KUKA KRL program: MyProgram_193().src

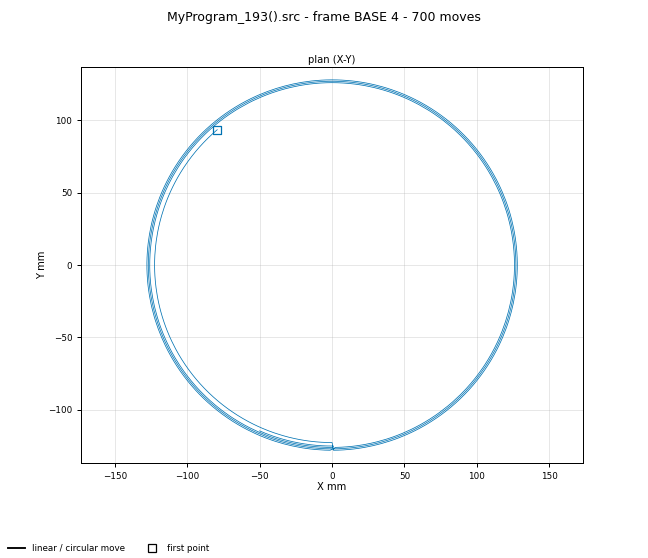
[picture p0: tool path of MyProgram_193().src in frame BASE 4, 700 of 700 moves have a stored position in this frame; points joined in program order, loops and branches not executed]
&ACCESS RVP
&REL 1
&PARAM TEMPLATE = C:\KRC\Roboter\Template\vorgabe
&PARAM EDITMASK = *
DEF MyProgram_193()
; ---- Setting reference (Base) ----
$BASE = BASE_DATA[4]

; --------------------------
; ---- Setting tool (TCP) ----
$TOOL = TOOL_DATA[3]
; --------------------------

$VEL.CP = VEL_APROX_PRINT
Startdeposition()
$VEL.CP = VEL_PRINT
LIN {X -79.3887,Y 93.5146,Z 139,A 127.081,B 23.6673,C -1.501,E1 23.6075,E2 679.4416} C_DIS
LIN {X -82.6375,Y 90.6569,Z 139,A 129.0803,B 23.6676,C -1.4955,E1 23.6034,E2 677.4477} C_DIS
LIN {X -85.6654,Y 87.8014,Z 139,A 131.1027,B 23.6676,C -1.4942,E1 23.5993,E2 675.4197} C_DIS
LIN {X -88.7871,Y 84.6429,Z 139,A 133.1305,B 23.6681,C -1.4871,E1 23.5954,E2 673.4002} C_DIS
LIN {X -91.627,Y 81.5608,Z 139,A 135.1651,B 23.6682,C -1.4854,E1 23.5916,E2 671.3603} C_DIS
LIN {X -94.341,Y 78.4052,Z 139,A 137.0999,B 23.6685,C -1.48,E1 23.5881,E2 669.4298} C_DIS
LIN {X -97.1692,Y 74.872,Z 139,A 139.2464,B 23.6688,C -1.4757,E1 23.5844,E2 667.2831} C_DIS
LIN {X -99.8211,Y 71.2973,Z 139,A 141.3446,B 23.6691,C -1.4708,E1 23.5809,E2 665.1863} C_DIS
LIN {X -102.4361,Y 67.4863,Z 139,A 143.4891,B 23.6694,C -1.4642,E1 23.5776,E2 663.047} C_DIS
LIN {X -104.8157,Y 63.7284,Z 139,A 145.6026,B 23.6697,C -1.4598,E1 23.5745,E2 660.9332} C_DIS
LIN {X -106.7407,Y 60.4493,Z 139,A 147.3793,B 23.67,C -1.4547,E1 23.572,E2 659.1594} C_DIS
LIN {X -108.6109,Y 57.0154,Z 139,A 149.1562,B 23.6704,C -1.4473,E1 23.5697,E2 657.391} C_DIS
LIN {X -110.2377,Y 53.8052,Z 139,A 150.913,B 23.6705,C -1.4454,E1 23.5675,E2 655.6289} C_DIS
LIN {X -111.8084,Y 50.4593,Z 139,A 152.53,B 23.6711,C -1.4356,E1 23.5657,E2 654.027} C_DIS
LIN {X -113.3266,Y 46.9501,Z 139,A 154.4547,B 23.6711,C -1.4359,E1 23.5636,E2 652.0901} C_DIS
LIN {X -114.6812,Y 43.5389,Z 139,A 156.1243,B 23.6715,C -1.4288,E1 23.5619,E2 650.4286} C_DIS
LIN {X -115.9983,Y 39.8949,Z 139,A 157.8402,B 23.672,C -1.4193,E1 23.5603,E2 648.7262} C_DIS
LIN {X -116.9413,Y 37.0399,Z 139,A 159.2538,B 23.6723,C -1.4152,E1 23.5591,E2 647.314} C_DIS
LIN {X -117.8141,Y 34.1624,Z 139,A 160.8056,B 23.6722,C -1.4169,E1 23.5578,E2 645.7485} C_DIS
LIN {X -118.9906,Y 29.8083,Z 139,A 162.938,B 23.6725,C -1.4113,E1 23.5563,E2 643.6172} C_DIS
LIN {X -119.8593,Y 26.095,Z 139,A 164.7128,B 23.6728,C -1.4053,E1 23.5553,E2 641.8462} C_DIS
LIN {X -120.5971,Y 22.4467,Z 139,A 166.3262,B 23.6734,C -1.3945,E1 23.5544,E2 640.2496} C_DIS
LIN {X -121.1103,Y 19.4926,Z 139,A 167.753,B 23.6736,C -1.3911,E1 23.5538,E2 638.8224} C_DIS
LIN {X -121.55,Y 16.5267,Z 139,A 169.2845,B 23.6736,C -1.392,E1 23.5532,E2 637.279} C_DIS
LIN {X -121.9936,Y 12.8387,Z 139,A 170.9072,B 23.6741,C -1.3817,E1 23.5527,E2 635.6716} C_DIS
LIN {X -122.2705,Y 9.8652,Z 139,A 172.3135,B 23.6743,C -1.3777,E1 23.5523,E2 634.2665} C_DIS
LIN {X -122.4784,Y 6.8343,Z 139,A 173.7573,B 23.6745,C -1.3741,E1 23.5521,E2 632.8224} C_DIS
LIN {X -122.6313,Y 2.9913,Z 139,A 175.5814,B 23.6748,C -1.3694,E1 23.5519,E2 630.9984} C_DIS
LIN {X -122.6672,Y -0.3879,Z 139,A 177.2488,B 23.6748,C -1.368,E1 23.5519,E2 629.324} C_DIS
LIN {X -122.5842,Y -4.5164,Z 139,A 179.0836,B 23.6754,C -1.3579,E1 23.552,E2 627.5027} C_DIS
LIN {X -122.44,Y -7.4601,Z 139,A -179.4399,B 23.6754,C -1.3576,E1 23.5523,E2 626.0175} C_DIS
LIN {X -122.1123,Y -11.6529,Z 139,A -177.4861,B 23.6758,C -1.3509,E1 23.5527,E2 624.0681} C_DIS
LIN {X -121.6563,Y -15.7152,Z 139,A -175.6057,B 23.6762,C -1.3436,E1 23.5534,E2 622.1941} C_DIS
LIN {X -121.2209,Y -18.7791,Z 139,A -174.1758,B 23.6765,C -1.3383,E1 23.5539,E2 620.7682} C_DIS
LIN {X -120.73,Y -21.7125,Z 139,A -172.7657,B 23.6767,C -1.3348,E1 23.5546,E2 619.358} C_DIS
LIN {X -120.0095,Y -25.3991,Z 139,A -170.9856,B 23.6769,C -1.3304,E1 23.5556,E2 617.5779} C_DIS
LIN {X -119.1851,Y -29.0196,Z 139,A -169.2623,B 23.6772,C -1.3246,E1 23.5567,E2 615.8584} C_DIS
LIN {X -118.4092,Y -32.0405,Z 139,A -167.6338,B 23.6771,C -1.3272,E1 23.5579,E2 614.2133} C_DIS
LIN {X -117.3595,Y -35.6921,Z 139,A -166.0055,B 23.6777,C -1.3157,E1 23.5592,E2 612.6037} C_DIS
LIN {X -116.2196,Y -39.248,Z 139,A -164.0849,B 23.6776,C -1.3178,E1 23.5608,E2 610.6662} C_DIS
LIN {X -114.9815,Y -42.7371,Z 139,A -162.5098,B 23.6782,C -1.3062,E1 23.5623,E2 609.1106} C_DIS
LIN {X -113.8941,Y -45.556,Z 139,A -160.9775,B 23.6782,C -1.3072,E1 23.5639,E2 607.567} C_DIS
LIN {X -112.4784,Y -48.9468,Z 139,A -159.3454,B 23.6786,C -1.2987,E1 23.5657,E2 605.9466} C_DIS
LIN {X -110.9144,Y -52.3963,Z 139,A -157.5959,B 23.6789,C -1.2928,E1 23.5677,E2 604.2016} C_DIS
LIN {X -109.5682,Y -55.1562,Z 139,A -156.145,B 23.679,C -1.2895,E1 23.5695,E2 602.7507} C_DIS
LIN {X -108.185,Y -57.824,Z 139,A -154.585,B 23.6789,C -1.2921,E1 23.5716,E2 601.1753} C_DIS
LIN {X -105.9858,Y -61.7632,Z 139,A -152.4677,B 23.6792,C -1.2868,E1 23.5745,E2 599.0594} C_DIS
LIN {X -104.0005,Y -65.0502,Z 139,A -150.6485,B 23.6793,C -1.2832,E1 23.5772,E2 597.2395} C_DIS
LIN {X -101.5455,Y -68.819,Z 139,A -148.5147,B 23.6796,C -1.2792,E1 23.5805,E2 595.1044} C_DIS
LIN {X -98.9417,Y -72.5127,Z 139,A -146.4248,B 23.6799,C -1.273,E1 23.5839,E2 593.0191} C_DIS
LIN {X -96.2459,Y -76.0552,Z 139,A -144.3049,B 23.68,C -1.2697,E1 23.5875,E2 590.8969} C_DIS
LIN {X -93.644,Y -79.2365,Z 139,A -142.5065,B 23.6805,C -1.26,E1 23.5907,E2 589.1139} C_DIS
LIN {X -91.1571,Y -82.0855,Z 139,A -140.6177,B 23.6805,C -1.2612,E1 23.5942,E2 587.2131} C_DIS
LIN {X -88.24,Y -85.2131,Z 139,A -138.6381,B 23.6807,C -1.256,E1 23.598,E2 585.2373} C_DIS
LIN {X -85.1287,Y -88.3217,Z 139,A -136.6069,B 23.681,C -1.2507,E1 23.6021,E2 583.2104} C_DIS
LIN {X -82.1159,Y -91.1299,Z 139,A -134.5975,B 23.681,C -1.2504,E1 23.6062,E2 581.193} C_DIS
LIN {X -78.7723,Y -94.0344,Z 139,A -132.6267,B 23.6814,C -1.2422,E1 23.6104,E2 579.2346} C_DIS
LIN {X -75.7059,Y -96.5203,Z 139,A -130.7809,B 23.6816,C -1.2389,E1 23.6144,E2 577.3898} C_DIS
LIN {X -72.5193,Y -98.9369,Z 139,A -128.955,B 23.6818,C -1.2338,E1 23.6185,E2 575.5698} C_DIS
LIN {X -69.4074,Y -101.1442,Z 139,A -127.0058,B 23.6816,C -1.238,E1 23.623,E2 573.6029} C_DIS
LIN {X -65.6311,Y -103.6346,Z 139,A -124.9026,B 23.6818,C -1.2343,E1 23.6279,E2 571.5018} C_DIS
LIN {X -61.7652,Y -105.9846,Z 139,A -122.7608,B 23.6818,C -1.2324,E1 23.6331,E2 569.3578} C_DIS
LIN {X -57.8305,Y -108.1816,Z 139,A -120.6273,B 23.682,C -1.2308,E1 23.6383,E2 567.2219} C_DIS
LIN {X -54.5438,Y -109.8734,Z 139,A -119.0576,B 23.6824,C -1.2218,E1 23.6422,E2 565.6702} C_DIS
LIN {X -51.5071,Y -111.3288,Z 139,A -117.4725,B 23.6824,C -1.2205,E1 23.6462,E2 564.0843} C_DIS
LIN {X -48.3233,Y -112.748,Z 139,A -115.7041,B 23.6823,C -1.2249,E1 23.6507,E2 562.3005} C_DIS
LIN {X -44.1464,Y -114.4478,Z 139,A -113.6361,B 23.6824,C -1.2211,E1 23.6561,E2 560.237} C_DIS
LIN {X -39.9096,Y -115.9932,Z 139,A -111.6551,B 23.6828,C -1.2137,E1 23.6613,E2 558.2704} C_DIS
LIN {X -37.055,Y -116.9364,Z 139,A -110.2492,B 23.6828,C -1.2126,E1 23.665,E2 556.8643} C_DIS
LIN {X -34.1778,Y -117.8096,Z 139,A -108.7044,B 23.6826,C -1.2179,E1 23.6692,E2 555.3038} C_DIS
LIN {X -29.8197,Y -118.9876,Z 139,A -106.5916,B 23.6826,C -1.2168,E1 23.6749,E2 553.1904} C_DIS
LIN {X -25.9912,Y -119.8817,Z 139,A -104.7935,B 23.6828,C -1.2142,E1 23.6798,E2 551.3964} C_DIS
LIN {X -22.4579,Y -120.595,Z 139,A -103.0548,B 23.6827,C -1.216,E1 23.6846,E2 549.6512} C_DIS
LIN {X -18.7973,Y -121.2181,Z 139,A -101.4495,B 23.683,C -1.2097,E1 23.6889,E2 548.0601} C_DIS
LIN {X -15.7039,Y -121.6578,Z 139,A -99.8752,B 23.6828,C -1.2145,E1 23.6933,E2 546.4724} C_DIS
LIN {X -11.2234,Y -122.1535,Z 139,A -97.7609,B 23.6828,C -1.2147,E1 23.6992,E2 544.3564} C_DIS
LIN {X -7.5226,Y -122.4362,Z 139,A -96.1117,B 23.6829,C -1.2109,E1 23.7038,E2 542.7161} C_DIS
LIN {X -3.7044,Y -122.6115,Z 139,A -94.259,B 23.6828,C -1.2141,E1 23.709,E2 540.855} C_DIS
LIN {X -0.005,Y -122.669,Z 139,A -92.6349,B 23.683,C -1.2097,E1 23.7135,E2 539.2418} C_DIS
LIN {X -0.005,Y -122.669,Z 139,A -92.6349,B 23.683,C -1.2097,E1 23.7135,E2 539.2418} C_DIS
Enddeposition()
LIN {X 0.9076,Y -127.9731,Z 140,A -92.6066,B 24.9649,C -1.3697,E1 25.0021,E2 539.0016} C_DIS
Startdeposition()
$VEL.CP = VEL_PRINT
LIN {X 4.2701,Y -127.9089,Z 140,A -90.8609,B 24.9642,C -1.3823,E1 25.0071,E2 537.2265} C_DIS
LIN {X 8.0025,Y -127.7277,Z 140,A -89.2685,B 24.9644,C -1.3789,E1 25.0115,E2 535.6426} C_DIS
LIN {X 12.0529,Y -127.4094,Z 140,A -87.5467,B 24.9646,C -1.3749,E1 25.0162,E2 533.9312} C_DIS
LIN {X 14.9814,Y -127.0982,Z 140,A -86.1517,B 24.9643,C -1.3796,E1 25.0201,E2 532.5262} C_DIS
LIN {X 18.2831,Y -126.6654,Z 140,A -84.6512,B 24.9643,C -1.3811,E1 25.0243,E2 531.0233} C_DIS
LIN {X 22.3408,Y -126.013,Z 140,A -82.8669,B 24.9643,C -1.3797,E1 25.0292,E2 529.2443} C_DIS
LIN {X 25.4642,Y -125.419,Z 140,A -81.4803,B 24.9643,C -1.379,E1 25.033,E2 527.8608} C_DIS
LIN {X 28.3673,Y -124.7944,Z 140,A -80.2161,B 24.9645,C -1.3769,E1 25.0364,E2 526.6033} C_DIS
LIN {X 31.3018,Y -124.0909,Z 140,A -78.771,B 24.9642,C -1.3831,E1 25.0404,E2 525.1456} C_DIS
LIN {X 34.2875,Y -123.2993,Z 140,A -77.4974,B 24.9644,C -1.379,E1 25.0438,E2 523.8838} C_DIS
LIN {X 37.2721,Y -122.4301,Z 140,A -76.2359,B 24.9646,C -1.3739,E1 25.0471,E2 522.6365} C_DIS
LIN {X 40.0928,Y -121.536,Z 140,A -74.6318,B 24.9638,C -1.3899,E1 25.0515,E2 520.9976} C_DIS
LIN {X 43.2265,Y -120.4567,Z 140,A -73.2401,B 24.964,C -1.3871,E1 25.0551,E2 519.6153} C_DIS
LIN {X 46.1903,Y -119.3515,Z 140,A -71.7808,B 24.9637,C -1.3913,E1 25.0589,E2 518.1492} C_DIS
LIN {X 49.1413,Y -118.1671,Z 140,A -70.3614,B 24.9637,C -1.3932,E1 25.0626,E2 516.7287} C_DIS
LIN {X 51.9549,Y -116.9576,Z 140,A -69.1813,B 24.964,C -1.3854,E1 25.0656,E2 515.5699} C_DIS
LIN {X 54.9013,Y -115.6037,Z 140,A -67.5632,B 24.9635,C -1.3963,E1 25.0697,E2 513.9301} C_DIS
LIN {X 57.8129,Y -114.1754,Z 140,A -66.0746,B 24.9633,C -1.4007,E1 25.0735,E2 512.4352} C_DIS
LIN {X 60.9283,Y -112.5463,Z 140,A -64.3996,B 24.9628,C -1.4087,E1 25.0776,E2 510.746} C_DIS
LIN {X 64.6643,Y -110.4415,Z 140,A -62.4971,B 24.9627,C -1.4113,E1 25.0822,E2 508.843} C_DIS
LIN {X 68.3933,Y -108.1717,Z 140,A -60.6188,B 24.9627,C -1.4111,E1 25.0867,E2 506.9712} C_DIS
LIN {X 71.8212,Y -105.9268,Z 140,A -58.7909,B 24.9625,C -1.4145,E1 25.0909,E2 505.1415} C_DIS
LIN {X 75.297,Y -103.4851,Z 140,A -56.8856,B 24.9623,C -1.4186,E1 25.0953,E2 503.233} C_DIS
LIN {X 78.6223,Y -100.982,Z 140,A -54.9796,B 24.962,C -1.425,E1 25.0995,E2 501.3189} C_DIS
LIN {X 81.9467,Y -98.3039,Z 140,A -53.0464,B 24.9617,C -1.4304,E1 25.1037,E2 499.3801} C_DIS
LIN {X 85.2482,Y -95.4543,Z 140,A -51.1346,B 24.9615,C -1.4329,E1 25.1077,E2 497.4702} C_DIS
LIN {X 88.4654,Y -92.4804,Z 140,A -49.1994,B 24.9614,C -1.4363,E1 25.1116,E2 495.535} C_DIS
LIN {X 91.6345,Y -89.3421,Z 140,A -47.1815,B 24.961,C -1.4424,E1 25.1156,E2 493.5112} C_DIS
LIN {X 94.5006,Y -86.305,Z 140,A -45.3542,B 24.9609,C -1.4449,E1 25.1191,E2 491.686} C_DIS
LIN {X 97.2409,Y -83.2054,Z 140,A -43.4679,B 24.9605,C -1.4516,E1 25.1225,E2 489.7924} C_DIS
LIN {X 100.0412,Y -79.8156,Z 140,A -41.547,B 24.9604,C -1.4544,E1 25.1259,E2 487.8738} C_DIS
LIN {X 102.646,Y -76.4365,Z 140,A -39.6801,B 24.9602,C -1.4574,E1 25.129,E2 486.0088} C_DIS
LIN {X 105.1099,Y -73.0114,Z 140,A -37.8242,B 24.96,C -1.461,E1 25.132,E2 484.1535} C_DIS
LIN {X 107.2878,Y -69.7717,Z 140,A -36.0336,B 24.9596,C -1.4683,E1 25.1348,E2 482.3546} C_DIS
LIN {X 109.6772,Y -65.9528,Z 140,A -34.1134,B 24.9596,C -1.469,E1 25.1376,E2 480.4424} C_DIS
LIN {X 111.6754,Y -62.5093,Z 140,A -32.2598,B 24.9591,C -1.4781,E1 25.1402,E2 478.5769} C_DIS
LIN {X 113.7807,Y -58.5882,Z 140,A -30.3362,B 24.9589,C -1.4805,E1 25.1427,E2 476.658} C_DIS
LIN {X 115.1293,Y -55.8943,Z 140,A -29.0433,B 24.9589,C -1.4816,E1 25.1443,E2 475.3694} C_DIS
LIN {X 116.4969,Y -52.9848,Z 140,A -27.6149,B 24.9587,C -1.4854,E1 25.1459,E2 473.9396} C_DIS
LIN {X 117.9777,Y -49.5948,Z 140,A -25.9435,B 24.9583,C -1.4914,E1 25.1478,E2 472.2632} C_DIS
LIN {X 119.233,Y -46.4952,Z 140,A -24.5,B 24.9583,C -1.4933,E1 25.1493,E2 470.8233} C_DIS
LIN {X 120.2222,Y -43.8768,Z 140,A -23.1739,B 24.9578,C -1.5011,E1 25.1506,E2 469.4861} C_DIS
LIN {X 121.1957,Y -41.1148,Z 140,A -21.8125,B 24.9574,C -1.508,E1 25.1518,E2 468.1162} C_DIS
LIN {X 122.3197,Y -37.6329,Z 140,A -20.3174,B 24.9575,C -1.5056,E1 25.1531,E2 466.6353} C_DIS
LIN {X 123.2027,Y -34.6331,Z 140,A -19.0434,B 24.9577,C -1.5034,E1 25.154,E2 465.3737} C_DIS
LIN {X 123.8556,Y -32.229,Z 140,A -17.7303,B 24.9569,C -1.5176,E1 25.155,E2 464.0348} C_DIS
LIN {X 124.5942,Y -29.2441,Z 140,A -16.3459,B 24.9566,C -1.5225,E1 25.1559,E2 462.6469} C_DIS
LIN {X 125.2565,Y -26.2628,Z 140,A -14.9625,B 24.9563,C -1.5278,E1 25.1567,E2 461.259} C_DIS
LIN {X 125.9442,Y -22.7253,Z 140,A -13.4705,B 24.9563,C -1.5266,E1 25.1574,E2 459.7785} C_DIS
LIN {X 126.4433,Y -19.761,Z 140,A -12.168,B 24.9563,C -1.5287,E1 25.158,E2 458.4787} C_DIS
LIN {X 126.8932,Y -16.6281,Z 140,A -10.7317,B 24.9559,C -1.5344,E1 25.1586,E2 457.0375} C_DIS
LIN {X 127.3223,Y -12.9601,Z 140,A -8.9614,B 24.9552,C -1.5461,E1 25.1591,E2 455.2501} C_DIS
LIN {X 127.6326,Y -9.3972,Z 140,A -7.5269,B 24.9554,C -1.5425,E1 25.1594,E2 453.8326} C_DIS
LIN {X 127.8325,Y -6.1114,Z 140,A -5.9091,B 24.9547,C -1.5551,E1 25.1597,E2 452.1947} C_DIS
LIN {X 127.9576,Y -2.3014,Z 140,A -4.346,B 24.9548,C -1.553,E1 25.1597,E2 450.6458} C_DIS
LIN {X 127.9704,Y 1.5309,Z 140,A -2.5591,B 24.9543,C -1.5624,E1 25.1597,E2 448.8473} C_DIS
LIN {X 127.8741,Y 5.1617,Z 140,A -1.0017,B 24.9542,C -1.5641,E1 25.1597,E2 447.2952} C_DIS
LIN {X 127.6513,Y 9.1421,Z 140,A 0.7262,B 24.954,C -1.5669,E1 25.1593,E2 445.5709} C_DIS
LIN {X 127.4094,Y 12.0529,Z 140,A 2.0613,B 24.9537,C -1.5727,E1 25.159,E2 444.2302} C_DIS
LIN {X 127.0363,Y 15.5009,Z 140,A 3.7184,B 24.953,C -1.5833,E1 25.1584,E2 442.5579} C_DIS
LIN {X 126.5623,Y 18.9921,Z 140,A 5.2467,B 24.9529,C -1.5857,E1 25.1578,E2 441.0329} C_DIS
LIN {X 126.0297,Y 22.2478,Z 140,A 6.6306,B 24.9529,C -1.5855,E1 25.1572,E2 439.6575} C_DIS
LIN {X 125.4446,Y 25.3382,Z 140,A 8.0006,B 24.9528,C -1.588,E1 25.1564,E2 438.2898} C_DIS
LIN {X 124.7727,Y 28.4626,Z 140,A 9.3377,B 24.9528,C -1.5875,E1 25.1556,E2 436.9615} C_DIS
LIN {X 124.0864,Y 31.3198,Z 140,A 10.7285,B 24.9523,C -1.5957,E1 25.1547,E2 435.5595} C_DIS
LIN {X 123.04,Y 35.2148,Z 140,A 12.5291,B 24.952,C -1.601,E1 25.1534,E2 433.7568} C_DIS
LIN {X 122.1223,Y 38.2746,Z 140,A 14.0391,B 24.9515,C -1.6097,E1 25.1521,E2 432.2349} C_DIS
LIN {X 120.9796,Y 41.7406,Z 140,A 15.5777,B 24.9515,C -1.6097,E1 25.1507,E2 430.705} C_DIS
LIN {X 119.9332,Y 44.6586,Z 140,A 16.9722,B 24.9512,C -1.6142,E1 25.1494,E2 429.3076} C_DIS
LIN {X 118.7692,Y 47.6676,Z 140,A 18.3953,B 24.951,C -1.6173,E1 25.1479,E2 427.885} C_DIS
LIN {X 117.5887,Y 50.5101,Z 140,A 19.5686,B 24.9514,C -1.6106,E1 25.1467,E2 426.7341} C_DIS
LIN {X 116.282,Y 53.4496,Z 140,A 21.2237,B 24.9505,C -1.6261,E1 25.1448,E2 425.0513} C_DIS
LIN {X 114.8656,Y 56.4288,Z 140,A 22.6722,B 24.9503,C -1.6289,E1 25.143,E2 423.604} C_DIS
LIN {X 113.3976,Y 59.3236,Z 140,A 24.1224,B 24.95,C -1.6328,E1 25.1412,E2 422.1522} C_DIS
LIN {X 111.366,Y 63.0599,Z 140,A 26.1237,B 24.9494,C -1.6432,E1 25.1384,E2 420.1368} C_DIS
LIN {X 109.3021,Y 66.5731,Z 140,A 27.9392,B 24.9491,C -1.6477,E1 25.1358,E2 418.32} C_DIS
LIN {X 107.0663,Y 70.1118,Z 140,A 29.8057,B 24.9488,C -1.6523,E1 25.133,E2 416.4521} C_DIS
LIN {X 104.6388,Y 73.685,Z 140,A 31.7003,B 24.9487,C -1.6552,E1 25.13,E2 414.5599} C_DIS
LIN {X 102.0732,Y 77.2,Z 140,A 33.6298,B 24.9484,C -1.6592,E1 25.1268,E2 412.6303} C_DIS
LIN {X 99.4073,Y 80.6043,Z 140,A 35.5612,B 24.9481,C -1.6637,E1 25.1234,E2 410.6974} C_DIS
LIN {X 96.7011,Y 83.8321,Z 140,A 37.495,B 24.9477,C -1.6706,E1 25.1199,E2 408.7559} C_DIS
LIN {X 93.9403,Y 86.9146,Z 140,A 39.2777,B 24.9477,C -1.6712,E1 25.1165,E2 406.9797} C_DIS
LIN {X 91.0503,Y 89.9374,Z 140,A 41.1467,B 24.9474,C -1.6752,E1 25.1129,E2 405.1093} C_DIS
LIN {X 88.1229,Y 92.8077,Z 140,A 43.0115,B 24.9471,C -1.6807,E1 25.1091,E2 403.2393} C_DIS
LIN {X 85.0157,Y 95.6619,Z 140,A 44.9026,B 24.9468,C -1.6847,E1 25.1052,E2 401.3464} C_DIS
LIN {X 81.942,Y 98.3079,Z 140,A 46.6565,B 24.9468,C -1.685,E1 25.1015,E2 399.5985} C_DIS
LIN {X 78.7277,Y 100.9003,Z 140,A 48.5386,B 24.9465,C -1.6902,E1 25.0974,E2 397.711} C_DIS
LIN {X 75.345,Y 103.4503,Z 140,A 50.4087,B 24.9463,C -1.6923,E1 25.0932,E2 395.8428} C_DIS
LIN {X 71.9763,Y 105.8218,Z 140,A 52.2755,B 24.9461,C -1.6966,E1 25.0889,E2 393.9722} C_DIS
LIN {X 68.0587,Y 108.3829,Z 140,A 54.3229,B 24.9461,C -1.6975,E1 25.0841,E2 391.9294} C_DIS
LIN {X 64.4713,Y 110.5548,Z 140,A 56.2279,B 24.9457,C -1.7017,E1 25.0795,E2 390.0203} C_DIS
LIN {X 60.7747,Y 112.6288,Z 140,A 58.1089,B 24.9457,C -1.7035,E1 25.0749,E2 388.1404} C_DIS
LIN {X 57.1568,Y 114.5065,Z 140,A 59.901,B 24.9456,C -1.7043,E1 25.0704,E2 386.3514} C_DIS
LIN {X 53.8901,Y 116.0783,Z 140,A 61.4268,B 24.9458,C -1.7013,E1 25.0666,E2 384.8365} C_DIS
LIN {X 50.0553,Y 117.7854,Z 140,A 63.433,B 24.9452,C -1.7099,E1 25.0614,E2 382.815} C_DIS
LIN {X 46.6151,Y 119.1864,Z 140,A 64.9753,B 24.9455,C -1.7055,E1 25.0575,E2 381.2865} C_DIS
LIN {X 43.5103,Y 120.3543,Z 140,A 66.2806,B 24.946,C -1.6978,E1 25.0541,E2 380.0021} C_DIS
LIN {X 41.1775,Y 121.1748,Z 140,A 67.6036,B 24.9452,C -1.7097,E1 25.0505,E2 378.6537} C_DIS
LIN {X 37.8444,Y 122.255,Z 140,A 69.164,B 24.9452,C -1.7105,E1 25.0464,E2 377.0941} C_DIS
LIN {X 34.5678,Y 123.2209,Z 140,A 70.6014,B 24.9454,C -1.707,E1 25.0425,E2 375.6674} C_DIS
LIN {X 30.3415,Y 124.3296,Z 140,A 72.4573,B 24.9456,C -1.7032,E1 25.0376,E2 373.8234} C_DIS
LIN {X 27.2217,Y 125.0495,Z 140,A 74.0505,B 24.9451,C -1.712,E1 25.0332,E2 372.2116} C_DIS
LIN {X 24.0369,Y 125.7003,Z 140,A 75.4916,B 24.9451,C -1.712,E1 25.0292,E2 370.7724} C_DIS
LIN {X 20.7847,Y 126.2792,Z 140,A 77.0061,B 24.9449,C -1.7142,E1 25.025,E2 369.254} C_DIS
LIN {X 16.8085,Y 126.8695,Z 140,A 78.7456,B 24.9451,C -1.7117,E1 25.0203,E2 367.522} C_DIS
LIN {X 13.7363,Y 127.2387,Z 140,A 80.1561,B 24.945,C -1.7132,E1 25.0163,E2 366.109} C_DIS
LIN {X 10.0436,Y 127.5855,Z 140,A 81.9323,B 24.9446,C -1.719,E1 25.0114,E2 364.3199} C_DIS
LIN {X 6.6351,Y 127.8062,Z 140,A 83.3074,B 24.9451,C -1.7114,E1 25.0076,E2 362.9633} C_DIS
LIN {X 3.3822,Y 127.9336,Z 140,A 84.8526,B 24.9448,C -1.7156,E1 25.0032,E2 361.4085} C_DIS
LIN {X -0.5369,Y 127.9772,Z 140,A 86.5777,B 24.945,C -1.7139,E1 24.9984,E2 359.6877} C_DIS
LIN {X -4.2701,Y 127.9089,Z 140,A 88.3434,B 24.9447,C -1.718,E1 24.9935,E2 357.9121} C_DIS
LIN {X -7.3727,Y 127.7665,Z 140,A 89.6721,B 24.9449,C -1.7144,E1 24.9898,E2 356.5914} C_DIS
LIN {X -10.6356,Y 127.5354,Z 140,A 91.1001,B 24.9451,C -1.712,E1 24.9858,E2 355.1686} C_DIS
LIN {X -14.425,Y 127.1646,Z 140,A 92.7573,B 24.9453,C -1.7087,E1 24.9813,E2 353.5182} C_DIS
LIN {X -17.9065,Y 126.7192,Z 140,A 94.2585,B 24.9456,C -1.7044,E1 24.9771,E2 352.0262} C_DIS
LIN {X -20.8827,Y 126.2628,Z 140,A 95.6821,B 24.9454,C -1.7071,E1 24.9732,E2 350.5949} C_DIS
LIN {X -23.8508,Y 125.7359,Z 140,A 97.0402,B 24.9454,C -1.7064,E1 24.9694,E2 349.2369} C_DIS
LIN {X -26.8272,Y 125.1346,Z 140,A 98.4043,B 24.9454,C -1.7055,E1 24.9657,E2 347.8734} C_DIS
LIN {X -29.8344,Y 124.4519,Z 140,A 99.7833,B 24.9456,C -1.7041,E1 24.962,E2 346.4958} C_DIS
LIN {X -32.7946,Y 123.7048,Z 140,A 101.1615,B 24.9456,C -1.7033,E1 24.9582,E2 345.1175} C_DIS
LIN {X -35.8577,Y 122.8518,Z 140,A 102.5709,B 24.9458,C -1.7011,E1 24.9545,E2 343.7112} C_DIS
LIN {X -38.6322,Y 122.0081,Z 140,A 103.9297,B 24.9457,C -1.7025,E1 24.9508,E2 342.3467} C_DIS
LIN {X -41.7684,Y 120.97,Z 140,A 105.389,B 24.9459,C -1.6997,E1 24.947,E2 340.8912} C_DIS
LIN {X -44.5407,Y 119.9773,Z 140,A 106.7502,B 24.9459,C -1.7,E1 24.9434,E2 339.5266} C_DIS
LIN {X -47.7395,Y 118.7402,Z 140,A 108.225,B 24.9462,C -1.695,E1 24.9396,E2 338.0604} C_DIS
LIN {X -50.3417,Y 117.6615,Z 140,A 109.554,B 24.9461,C -1.6964,E1 24.9362,E2 336.7251} C_DIS
LIN {X -53.2438,Y 116.3772,Z 140,A 110.8221,B 24.9467,C -1.6869,E1 24.933,E2 335.4765} C_DIS
LIN {X -56.2714,Y 114.9433,Z 140,A 112.4688,B 24.9464,C -1.6915,E1 24.9288,E2 333.8146} C_DIS
LIN {X -59.3236,Y 113.3976,Z 140,A 113.9543,B 24.9467,C -1.6867,E1 24.9251,E2 332.3363} C_DIS
LIN {X -62.81,Y 111.5064,Z 140,A 115.8077,B 24.9467,C -1.6873,E1 24.9206,E2 330.4764} C_DIS
LIN {X -66.4172,Y 109.3963,Z 140,A 117.7249,B 24.9467,C -1.686,E1 24.916,E2 328.5563} C_DIS
LIN {X -70.0382,Y 107.1147,Z 140,A 119.7053,B 24.9467,C -1.6853,E1 24.9113,E2 326.5711} C_DIS
LIN {X -73.5809,Y 104.7122,Z 140,A 121.6148,B 24.947,C -1.6811,E1 24.9069,E2 324.6652} C_DIS
LIN {X -77.1713,Y 102.0948,Z 140,A 123.5505,B 24.9475,C -1.6744,E1 24.9026,E2 322.7387} C_DIS
LIN {X -80.4221,Y 99.5542,Z 140,A 125.3987,B 24.9477,C -1.6704,E1 24.8986,E2 320.8931} C_DIS
LIN {X -83.5947,Y 96.9056,Z 140,A 127.2585,B 24.9479,C -1.6666,E1 24.8946,E2 319.035} C_DIS
LIN {X -86.6873,Y 94.1492,Z 140,A 129.122,B 24.9482,C -1.6627,E1 24.8908,E2 317.1735} C_DIS
LIN {X -89.684,Y 91.2991,Z 140,A 130.9841,B 24.9484,C -1.6587,E1 24.887,E2 315.3131} C_DIS
LIN {X -92.5909,Y 88.3497,Z 140,A 132.8534,B 24.9487,C -1.6548,E1 24.8834,E2 313.4451} C_DIS
LIN {X -95.4919,Y 85.2062,Z 140,A 134.8134,B 24.9489,C -1.652,E1 24.8797,E2 311.4831} C_DIS
LIN {X -98.3241,Y 81.9224,Z 140,A 136.7747,B 24.9491,C -1.6478,E1 24.8762,E2 309.5228} C_DIS
LIN {X -100.9003,Y 78.7277,Z 140,A 138.6622,B 24.9493,C -1.6451,E1 24.8729,E2 307.6326} C_DIS
LIN {X -103.4625,Y 75.3282,Z 140,A 140.5726,B 24.9496,C -1.6401,E1 24.8697,E2 305.7251} C_DIS
LIN {X -106.0437,Y 71.6484,Z 140,A 142.5286,B 24.9501,C -1.6318,E1 24.8666,E2 303.7792} C_DIS
LIN {X -108.3591,Y 68.0965,Z 140,A 144.4735,B 24.9503,C -1.6285,E1 24.8637,E2 301.8322} C_DIS
LIN {X -110.5548,Y 64.4713,Z 140,A 146.3991,B 24.9506,C -1.6243,E1 24.861,E2 299.9069} C_DIS
LIN {X -112.5462,Y 60.9283,Z 140,A 148.2396,B 24.9508,C -1.6198,E1 24.8585,E2 298.0672} C_DIS
LIN {X -114.4159,Y 57.3405,Z 140,A 149.9697,B 24.9514,C -1.6106,E1 24.8563,E2 296.3499} C_DIS
LIN {X -116.0186,Y 54.0192,Z 140,A 151.6307,B 24.9517,C -1.606,E1 24.8543,E2 294.6907} C_DIS
LIN {X -117.7854,Y 50.0553,Z 140,A 153.653,B 24.9518,C -1.6037,E1 24.8521,E2 292.6629} C_DIS
LIN {X -119.1516,Y 46.7046,Z 140,A 155.2204,B 24.9523,C -1.5962,E1 24.8505,E2 291.1045} C_DIS
LIN {X -120.3018,Y 43.6561,Z 140,A 156.5299,B 24.9529,C -1.5847,E1 24.8492,E2 289.815} C_DIS
LIN {X -121.2998,Y 40.8021,Z 140,A 158.0572,B 24.9527,C -1.5884,E1 24.8478,E2 288.2701} C_DIS
LIN {X -122.1466,Y 38.1986,Z 140,A 159.237,B 24.9531,C -1.5824,E1 24.8468,E2 287.0981} C_DIS
LIN {X -123.1836,Y 34.7013,Z 140,A 160.9106,B 24.9533,C -1.579,E1 24.8455,E2 285.4227} C_DIS
LIN {X -124.3118,Y 30.4156,Z 140,A 162.933,B 24.9536,C -1.5744,E1 24.8441,E2 283.3996} C_DIS
LIN {X -125.0286,Y 27.3181,Z 140,A 164.1866,B 24.9543,C -1.5619,E1 24.8434,E2 282.1684} C_DIS
LIN {X -125.6619,Y 24.2378,Z 140,A 165.7268,B 24.9543,C -1.5634,E1 24.8425,E2 280.6155} C_DIS
LIN {X -126.2167,Y 21.1594,Z 140,A 167.1076,B 24.9545,C -1.5579,E1 24.8418,E2 279.2396} C_DIS
LIN {X -126.6966,Y 18.0649,Z 140,A 168.4879,B 24.9549,C -1.5523,E1 24.8413,E2 277.8644} C_DIS
LIN {X -127.0621,Y 15.2845,Z 140,A 169.7862,B 24.9549,C -1.5502,E1 24.8408,E2 276.5635} C_DIS
LIN {X -127.3821,Y 12.3363,Z 140,A 171.1888,B 24.955,C -1.5493,E1 24.8404,E2 275.1546} C_DIS
LIN {X -127.6914,Y 8.5924,Z 140,A 172.888,B 24.9553,C -1.5445,E1 24.8401,E2 273.4565} C_DIS
LIN {X -127.8741,Y 5.1617,Z 140,A 174.4403,B 24.9556,C -1.5401,E1 24.8399,E2 271.9053} C_DIS
LIN {X -127.9723,Y 1.4172,Z 140,A 176.0883,B 24.956,C -1.5332,E1 24.8398,E2 270.2638} C_DIS
LIN {X -127.9536,Y -2.5439,Z 140,A 177.9563,B 24.956,C -1.5318,E1 24.8398,E2 268.3879} C_DIS
LIN {X -127.8255,Y -6.2512,Z 140,A 179.581,B 24.9564,C -1.5247,E1 24.84,E2 266.7703} C_DIS
LIN {X -127.5834,Y -10.0675,Z 140,A -178.5933,B 24.9564,C -1.5244,E1 24.8404,E2 264.9345} C_DIS
LIN {X -127.2627,Y -13.5137,Z 140,A -177.1468,B 24.957,C -1.5146,E1 24.8408,E2 263.5027} C_DIS
LIN {X -126.8695,Y -16.8085,Z 140,A -175.6162,B 24.9572,C -1.5119,E1 24.8413,E2 261.9694} C_DIS
LIN {X -126.2628,Y -20.8827,Z 140,A -173.8309,B 24.9577,C -1.5032,E1 24.8421,E2 260.1941} C_DIS
LIN {X -125.7359,Y -23.8508,Z 140,A -172.4692,B 24.9579,C -1.4995,E1 24.8428,E2 258.8333} C_DIS
LIN {X -125.1345,Y -26.8277,Z 140,A -171.0613,B 24.9579,C -1.4974,E1 24.8436,E2 257.422} C_DIS
LIN {X -124.4947,Y -29.6568,Z 140,A -169.7473,B 24.9582,C -1.494,E1 24.8444,E2 256.1083} C_DIS
LIN {X -123.6844,Y -32.8711,Z 140,A -168.3119,B 24.9586,C -1.4871,E1 24.8454,E2 254.681} C_DIS
LIN {X -122.8897,Y -35.7281,Z 140,A -166.9404,B 24.9586,C -1.485,E1 24.8465,E2 253.3066} C_DIS
LIN {X -122.113,Y -38.3039,Z 140,A -165.7853,B 24.959,C -1.479,E1 24.8474,E2 252.1591} C_DIS
LIN {X -121.0229,Y -41.6156,Z 140,A -164.1324,B 24.959,C -1.4786,E1 24.8489,E2 250.4979} C_DIS
LIN {X -120.1242,Y -44.1485,Z 140,A -162.83,B 24.959,C -1.4795,E1 24.8502,E2 249.1858} C_DIS
LIN {X -118.7692,Y -47.6676,Z 140,A -161.2539,B 24.9596,C -1.4693,E1 24.8518,E2 247.6252} C_DIS
LIN {X -117.6394,Y -50.393,Z 140,A -159.9724,B 24.9599,C -1.4636,E1 24.8531,E2 246.3503} C_DIS
LIN {X -116.2692,Y -53.4774,Z 140,A -158.3844,B 24.9599,C -1.4628,E1 24.855,E2 244.7555} C_DIS
LIN {X -115.1293,Y -55.8943,Z 140,A -157.1965,B 24.9601,C -1.4589,E1 24.8564,E2 243.5704} C_DIS
LIN {X -113.4456,Y -59.2322,Z 140,A -155.5103,B 24.9604,C -1.4548,E1 24.8586,E2 241.8849} C_DIS
LIN {X -111.6134,Y -62.6197,Z 140,A -153.6884,B 24.9604,C -1.4546,E1 24.861,E2 240.0539} C_DIS
LIN {X -109.4621,Y -66.3085,Z 140,A -151.805,B 24.9607,C -1.4481,E1 24.8637,E2 238.1764} C_DIS
LIN {X -107.2306,Y -69.8599,Z 140,A -149.9338,B 24.961,C -1.4428,E1 24.8665,E2 236.3083} C_DIS
LIN {X -104.8992,Y -73.3143,Z 140,A -147.987,B 24.961,C -1.4418,E1 24.8696,E2 234.3542} C_DIS
LIN {X -102.4032,Y -76.7626,Z 140,A -146.0493,B 24.9612,C -1.4385,E1 24.8728,E2 232.415} C_DIS
LIN {X -99.8763,Y -80.0228,Z 140,A -144.231,B 24.9616,C -1.4326,E1 24.876,E2 230.602} C_DIS
LIN {X -97.2409,Y -83.2054,Z 140,A -142.3323,B 24.9616,C -1.4306,E1 24.8794,E2 228.6995} C_DIS
LIN {X -94.5006,Y -86.305,Z 140,A -140.5093,B 24.962,C -1.4249,E1 24.8828,E2 226.8819} C_DIS
LIN {X -91.6287,Y -89.348,Z 140,A -138.6391,B 24.9622,C -1.4206,E1 24.8864,E2 225.0138} C_DIS
LIN {X -88.7217,Y -92.2355,Z 140,A -136.7844,B 24.9624,C -1.4177,E1 24.8901,E2 223.1584} C_DIS
LIN {X -85.6772,Y -95.0701,Z 140,A -134.8807,B 24.9624,C -1.4158,E1 24.894,E2 221.2514} C_DIS
LIN {X -82.545,Y -97.8019,Z 140,A -133.0013,B 24.9626,C -1.4131,E1 24.898,E2 219.3712} C_DIS
LIN {X -79.2656,Y -100.4778,Z 140,A -131.0944,B 24.9628,C -1.4101,E1 24.9022,E2 217.4643} C_DIS
LIN {X -75.5714,Y -103.2849,Z 140,A -129.0776,B 24.9631,C -1.4035,E1 24.9067,E2 215.456} C_DIS
LIN {X -72.0787,Y -105.7525,Z 140,A -127.14,B 24.9632,C -1.4014,E1 24.9111,E2 213.5168} C_DIS
LIN {X -68.6282,Y -108.0235,Z 140,A -125.2707,B 24.9633,C -1.3994,E1 24.9155,E2 211.6462} C_DIS
LIN {X -65.174,Y -110.142,Z 140,A -123.4007,B 24.9633,C -1.3994,E1 24.92,E2 209.7706} C_DIS
LIN {X -61.4342,Y -112.2703,Z 140,A -121.5242,B 24.9636,C -1.3942,E1 24.9245,E2 207.9008} C_DIS
LIN {X -58.5055,Y -113.8228,Z 140,A -120.0829,B 24.9638,C -1.3902,E1 24.9281,E2 206.4651} C_DIS
LIN {X -55.5481,Y -115.2947,Z 140,A -118.7523,B 24.9643,C -1.3812,E1 24.9314,E2 205.1525} C_DIS
LIN {X -52.9848,Y -116.4969,Z 140,A -117.2594,B 24.9638,C -1.3907,E1 24.9352,E2 203.6334} C_DIS
LIN {X -49.6385,Y -117.9594,Z 140,A -115.697,B 24.964,C -1.3854,E1 24.9392,E2 202.0799} C_DIS
LIN {X -46.6251,Y -119.1825,Z 140,A -114.2617,B 24.9642,C -1.3829,E1 24.9429,E2 200.6473} C_DIS
LIN {X -42.6642,Y -120.6594,Z 140,A -112.2382,B 24.9639,C -1.3876,E1 24.9483,E2 198.6085} C_DIS
LIN {X -39.1243,Y -121.8509,Z 140,A -110.7242,B 24.9644,C -1.3785,E1 24.9523,E2 197.1135} C_DIS
LIN {X -36.0788,Y -122.787,Z 140,A -109.2961,B 24.9644,C -1.3775,E1 24.9561,E2 195.6852} C_DIS
LIN {X -33.4495,Y -123.5302,Z 140,A -108.0086,B 24.9644,C -1.3799,E1 24.9596,E2 194.3901} C_DIS
LIN {X -30.1437,Y -124.3773,Z 140,A -106.6218,B 24.9647,C -1.3721,E1 24.9633,E2 193.0199} C_DIS
LIN {X -27.4685,Y -124.9962,Z 140,A -105.2226,B 24.9643,C -1.3799,E1 24.9672,E2 191.6004} C_DIS
LIN {X -24.1912,Y -125.6708,Z 140,A -103.8178,B 24.9646,C -1.3746,E1 24.971,E2 190.2065} C_DIS
LIN {X -21.1769,Y -126.2137,Z 140,A -102.4412,B 24.9646,C -1.3744,E1 24.9748,E2 188.8289} C_DIS
LIN {X -18.2831,Y -126.6654,Z 140,A -101.1007,B 24.9646,C -1.3756,E1 24.9785,E2 187.4847} C_DIS
LIN {X -14.9814,Y -127.0982,Z 140,A -99.5829,B 24.9646,C -1.3766,E1 24.9827,E2 185.9632} C_DIS
LIN {X -10.948,Y -127.5091,Z 140,A -98.0529,B 24.9652,C -1.3622,E1 24.9869,E2 184.4667} C_DIS
LIN {X -8.0445,Y -127.7251,Z 140,A -96.5808,B 24.9648,C -1.3706,E1 24.991,E2 182.974} C_DIS
LIN {X -4.9686,Y -127.8817,Z 140,A -95.0857,B 24.9645,C -1.3766,E1 24.9952,E2 181.4644} C_DIS
LIN {X -1.4172,Y -127.9723,Z 140,A -93.4122,B 24.9643,C -1.381,E1 24.9999,E2 179.7802} C_DIS
LIN {X -1.4172,Y -127.9723,Z 140,A -93.4122,B 24.9643,C -1.381,E1 24.9999,E2 179.7802} C_DIS
Enddeposition()
LIN {X 0.8984,Y -126.9978,Z 140,A -92.7232,B 24.9643,C -1.3809,E1 25.0018,E2 179.0917} C_DIS
Startdeposition()
$VEL.CP = VEL_PRINT
LIN {X -1.8864,Y -126.9894,Z 140,A -94.4585,B 24.9655,C -1.3568,E1 24.9968,E2 180.884} C_DIS
LIN {X -5.4454,Y -126.8874,Z 140,A -96.0999,B 24.9656,C -1.3549,E1 24.9922,E2 182.5303} C_DIS
LIN {X -9.0041,Y -126.6838,Z 140,A -97.7406,B 24.9656,C -1.3532,E1 24.9877,E2 184.1754} C_DIS
LIN {X -13.1754,Y -126.3185,Z 140,A -99.5978,B 24.9656,C -1.355,E1 24.9825,E2 186.0295} C_DIS
LIN {X -16.7396,Y -125.8953,Z 140,A -101.2605,B 24.9657,C -1.3531,E1 24.9779,E2 187.6978} C_DIS
LIN {X -20.7594,Y -125.295,Z 140,A -103.0018,B 24.9654,C -1.3582,E1 24.9731,E2 189.4287} C_DIS
LIN {X -24.376,Y -124.6429,Z 140,A -104.7874,B 24.9657,C -1.3526,E1 24.9682,E2 191.2295} C_DIS
LIN {X -27.9256,Y -123.8952,Z 140,A -106.4022,B 24.9657,C -1.3544,E1 24.9638,E2 192.842} C_DIS
LIN {X -31.9732,Y -122.9146,Z 140,A -108.2919,B 24.9657,C -1.3549,E1 24.9586,E2 194.7331} C_DIS
LIN {X -35.3331,Y -121.9895,Z 140,A -109.7594,B 24.9653,C -1.3611,E1 24.9547,E2 196.1883} C_DIS
LIN {X -38.5365,Y -121.0151,Z 140,A -111.2385,B 24.9652,C -1.3637,E1 24.9508,E2 197.6636} C_DIS
LIN {X -41.1445,Y -120.1544,Z 140,A -112.3647,B 24.9648,C -1.3702,E1 24.9479,E2 198.7766} C_DIS
LIN {X -45.1549,Y -118.7062,Z 140,A -114.2942,B 24.9648,C -1.3716,E1 24.9428,E2 200.7066} C_DIS
LIN {X -52.6173,Y -115.5927,Z 140,A -118.1702,B 24.9651,C -1.3645,E1 24.9328,E2 204.6085} C_DIS
LIN {X -55.96,Y -114.0097,Z 140,A -119.742,B 24.9648,C -1.3712,E1 24.9288,E2 206.1685} C_DIS
LIN {X -58.959,Y -112.4879,Z 140,A -121.532,B 24.9653,C -1.3602,E1 24.9243,E2 207.9895} C_DIS
LIN {X -63.3936,Y -110.0522,Z 140,A -123.6833,B 24.9649,C -1.3696,E1 24.9191,E2 210.1246} C_DIS
LIN {X -65.8137,Y -108.6219,Z 140,A -125.4418,B 24.9659,C -1.3484,E1 24.9148,E2 211.9389} C_DIS
LIN {X -69.7081,Y -106.1648,Z 140,A -127.0366,B 24.9646,C -1.3744,E1 24.9112,E2 213.4772} C_DIS
LIN {X -73.5077,Y -103.5708,Z 140,A -129.1354,B 24.9645,C -1.3768,E1 24.9064,E2 215.5775} C_DIS
LIN {X -76.7576,Y -101.1856,Z 140,A -130.9585,B 24.9643,C -1.3799,E1 24.9023,E2 217.3998} C_DIS
LIN {X -80.2298,Y -98.4548,Z 140,A -132.9521,B 24.9641,C -1.3836,E1 24.898,E2 219.3921} C_DIS
LIN {X -83.6741,Y -95.545,Z 140,A -134.984,B 24.9639,C -1.3877,E1 24.8937,E2 221.422} C_DIS
LIN {X -86.8883,Y -92.6321,Z 140,A -136.9403,B 24.9637,C -1.3917,E1 24.8896,E2 223.3767} C_DIS
LIN {X -89.9139,Y -89.6979,Z 140,A -138.8773,B 24.9636,C -1.3942,E1 24.8858,E2 225.316} C_DIS
LIN {X -93.0877,Y -86.3995,Z 140,A -141.003,B 24.9635,C -1.396,E1 24.8817,E2 227.4467} C_DIS
LIN {X -96.1754,Y -82.9484,Z 140,A -143.0221,B 24.9631,C -1.4041,E1 24.878,E2 229.4556} C_DIS
LIN {X -98.9796,Y -79.5816,Z 140,A -145.0005,B 24.9628,C -1.4087,E1 24.8745,E2 231.4321} C_DIS
LIN {X -100.9323,Y -77.0897,Z 140,A -146.4319,B 24.9626,C -1.4121,E1 24.8721,E2 232.8622} C_DIS
LIN {X -103.4983,Y -73.6095,Z 140,A -148.4617,B 24.9626,C -1.4134,E1 24.8687,E2 234.8988} C_DIS
LIN {X -105.9776,Y -69.9924,Z 140,A -150.3654,B 24.9621,C -1.422,E1 24.8658,E2 236.7916} C_DIS
LIN {X -108.1968,Y -66.5103,Z 140,A -152.282,B 24.962,C -1.4245,E1 24.8629,E2 238.712} C_DIS
LIN {X -110.5082,Y -62.5959,Z 140,A -154.3762,B 24.9618,C -1.4281,E1 24.86,E2 240.8085} C_DIS
LIN {X -112.8989,Y -58.1712,Z 140,A -156.4435,B 24.961,C -1.4437,E1 24.8573,E2 242.8496} C_DIS
LIN {X -114.2494,Y -55.4741,Z 140,A -157.9604,B 24.9611,C -1.4404,E1 24.8554,E2 244.3825} C_DIS
LIN {X -115.6893,Y -52.4025,Z 140,A -159.5393,B 24.9611,C -1.4426,E1 24.8536,E2 245.9648} C_DIS
LIN {X -117.1101,Y -49.1422,Z 140,A -161.0473,B 24.9605,C -1.4518,E1 24.8519,E2 247.4593} C_DIS
LIN {X -118.3429,Y -46.0941,Z 140,A -162.4702,B 24.9601,C -1.4589,E1 24.8505,E2 248.8731} C_DIS
LIN {X -119.4605,Y -43.115,Z 140,A -163.9244,B 24.9599,C -1.4624,E1 24.8491,E2 250.3273} C_DIS
LIN {X -120.4734,Y -40.198,Z 140,A -165.4088,B 24.9599,C -1.4624,E1 24.8477,E2 251.82} C_DIS
LIN {X -121.643,Y -36.5126,Z 140,A -167.8285,B 24.9613,C -1.4373,E1 24.8457,E2 254.3135} C_DIS
LIN {X -122.9805,Y -31.7137,Z 140,A -169.4765,B 24.9594,C -1.4713,E1 24.8446,E2 255.8901} C_DIS
LIN {X -123.6793,Y -28.8711,Z 140,A -171.39,B 24.9607,C -1.4488,E1 24.8434,E2 257.8685} C_DIS
LIN {X -124.6852,Y -24.1549,Z 140,A -172.9926,B 24.9589,C -1.4814,E1 24.8425,E2 259.4027} C_DIS
LIN {X -125.419,Y -20.0045,Z 140,A -174.955,B 24.9587,C -1.4848,E1 24.8416,E2 261.3689} C_DIS
LIN {X -125.9452,Y -16.3581,Z 140,A -176.5259,B 24.9582,C -1.4943,E1 24.841,E2 262.9265} C_DIS
LIN {X -126.3903,Y -12.4657,Z 140,A -178.4334,B 24.9582,C -1.4937,E1 24.8404,E2 264.8469} C_DIS
LIN {X -126.7622,Y -7.8201,Z 140,A 179.5644,B 24.9576,C -1.505,E1 24.84,E2 266.834} C_DIS
LIN {X -126.9481,Y -3.7458,Z 140,A 177.691,B 24.9573,C -1.5096,E1 24.8398,E2 268.7079} C_DIS
LIN {X -127.0052,Y -0.3954,Z 140,A 175.9852,B 24.9575,C -1.5057,E1 24.8398,E2 270.4331} C_DIS
LIN {X -126.9371,Y 4.1436,Z 140,A 174.0431,B 24.9569,C -1.5172,E1 24.8399,E2 272.3595} C_DIS
LIN {X -126.7555,Y 7.9289,Z 140,A 172.4083,B 24.9564,C -1.5263,E1 24.8402,E2 273.9826} C_DIS
LIN {X -126.46,Y 11.7393,Z 140,A 170.5524,B 24.9564,C -1.526,E1 24.8406,E2 275.8503} C_DIS
LIN {X -125.9639,Y 16.2156,Z 140,A 168.5002,B 24.956,C -1.5318,E1 24.8413,E2 277.901} C_DIS
LIN {X -125.3317,Y 20.539,Z 140,A 166.6266,B 24.9554,C -1.5426,E1 24.8421,E2 279.7599} C_DIS
LIN {X -124.7597,Y 23.7648,Z 140,A 165.1328,B 24.9552,C -1.5467,E1 24.8428,E2 281.2527} C_DIS
LIN {X -123.9228,Y 27.8051,Z 140,A 163.2886,B 24.9548,C -1.5536,E1 24.8439,E2 283.0915} C_DIS
LIN {X -123.2252,Y 30.7497,Z 140,A 161.8886,B 24.9546,C -1.5564,E1 24.8448,E2 284.493} C_DIS
LIN {X -122.3154,Y 34.1858,Z 140,A 160.4652,B 24.9538,C -1.5697,E1 24.8459,E2 285.8928} C_DIS
LIN {X -120.5823,Y 39.871,Z 140,A 157.589,B 24.9538,C -1.5695,E1 24.8483,E2 288.7862} C_DIS
LIN {X -119.497,Y 43.0135,Z 140,A 156.1023,B 24.9535,C -1.5748,E1 24.8496,E2 290.2686} C_DIS
LIN {X -118.0285,Y 46.8973,Z 140,A 154.1295,B 24.9535,C -1.5762,E1 24.8516,E2 292.2493} C_DIS
LIN {X -116.3531,Y 50.9113,Z 140,A 151.9144,B 24.9538,C -1.5709,E1 24.8541,E2 294.4892} C_DIS
LIN {X -114.9929,Y 53.9143,Z 140,A 150.6817,B 24.9528,C -1.5869,E1 24.8555,E2 295.6905} C_DIS
LIN {X -113.3654,Y 57.255,Z 140,A 149.0142,B 24.9525,C -1.5924,E1 24.8576,E2 297.3539} C_DIS
LIN {X -111.7153,Y 60.4149,Z 140,A 147.6185,B 24.9516,C -1.6068,E1 24.8594,E2 298.7226} C_DIS
LIN {X -109.9215,Y 63.6194,Z 140,A 145.5317,B 24.9525,C -1.5922,E1 24.8623,E2 300.8551} C_DIS
LIN {X -107.2101,Y 68.0902,Z 140,A 143.2675,B 24.9518,C -1.6033,E1 24.8656,E2 303.1043} C_DIS
LIN {X -104.8539,Y 71.665,Z 140,A 141.3529,B 24.9515,C -1.6096,E1 24.8686,E2 305.0137} C_DIS
LIN {X -102.4475,Y 75.0645,Z 140,A 139.4702,B 24.9511,C -1.6147,E1 24.8717,E2 306.8934} C_DIS
LIN {X -99.8336,Y 78.5074,Z 140,A 137.5017,B 24.9509,C -1.6191,E1 24.875,E2 308.8606} C_DIS
LIN {X -97.0222,Y 81.9572,Z 140,A 135.4519,B 24.9507,C -1.6225,E1 24.8787,E2 310.9117} C_DIS
LIN {X -94.1552,Y 85.2348,Z 140,A 133.5109,B 24.9503,C -1.6287,E1 24.8823,E2 312.8468} C_DIS
LIN {X -91.0647,Y 88.5293,Z 140,A 131.4498,B 24.95,C -1.6328,E1 24.8862,E2 314.9071} C_DIS
LIN {X -88.0521,Y 91.5267,Z 140,A 129.4938,B 24.9499,C -1.6357,E1 24.8901,E2 316.8645} C_DIS
LIN {X -84.8715,Y 94.4829,Z 140,A 127.5488,B 24.9495,C -1.6409,E1 24.8941,E2 318.8047} C_DIS
LIN {X -81.442,Y 97.4546,Z 140,A 125.5005,B 24.9493,C -1.6455,E1 24.8985,E2 320.8501} C_DIS
LIN {X -78.2125,Y 100.0652,Z 140,A 123.6055,B 24.9491,C -1.6487,E1 24.9026,E2 322.7447} C_DIS
LIN {X -74.8275,Y 102.6213,Z 140,A 121.6774,B 24.9489,C -1.6521,E1 24.9069,E2 324.6715} C_DIS
LIN {X -71.2998,Y 105.1024,Z 140,A 119.7407,B 24.9486,C -1.6564,E1 24.9114,E2 326.6044} C_DIS
LIN {X -67.5033,Y 107.5806,Z 140,A 117.663,B 24.9484,C -1.6589,E1 24.9163,E2 328.6829} C_DIS
LIN {X -63.9598,Y 109.7244,Z 140,A 115.6608,B 24.9486,C -1.6561,E1 24.9211,E2 330.6977} C_DIS
LIN {X -59.6983,Y 112.0996,Z 140,A 113.5726,B 24.948,C -1.6652,E1 24.9262,E2 332.7703} C_DIS
LIN {X -56.4433,Y 113.7713,Z 140,A 112.0707,B 24.9474,C -1.6749,E1 24.9299,E2 334.2532} C_DIS
LIN {X -53.6219,Y 115.1282,Z 140,A 110.659,B 24.9473,C -1.6772,E1 24.9335,E2 335.6631} C_DIS
LIN {X -49.781,Y 116.8418,Z 140,A 108.6004,B 24.9476,C -1.6724,E1 24.9388,E2 337.7377} C_DIS
LIN {X -46.3821,Y 118.2309,Z 140,A 107.0852,B 24.947,C -1.6814,E1 24.9426,E2 339.235} C_DIS
LIN {X -41.5699,Y 120.0069,Z 140,A 105.0533,B 24.946,C -1.6977,E1 24.9479,E2 341.2323} C_DIS
LIN {X -35.33,Y 121.9904,Z 140,A 101.6498,B 24.9471,C -1.6799,E1 24.9571,E2 344.6841} C_DIS
LIN {X -31.2642,Y 123.0946,Z 140,A 99.8747,B 24.9466,C -1.6878,E1 24.9618,E2 346.4431} C_DIS
LIN {X -28.3504,Y 123.7982,Z 140,A 98.5177,B 24.9466,C -1.6888,E1 24.9655,E2 347.7995} C_DIS
LIN {X -24.4459,Y 124.6295,Z 140,A 96.6595,B 24.9466,C -1.6876,E1 24.9706,E2 349.6627} C_DIS
LIN {X -21.1313,Y 125.2329,Z 140,A 95.1781,B 24.9464,C -1.6906,E1 24.9747,E2 351.1385} C_DIS
LIN {X -17.5614,Y 125.7837,Z 140,A 93.4456,B 24.9467,C -1.6868,E1 24.9795,E2 352.8814} C_DIS
LIN {X -13.5406,Y 126.2792,Z 140,A 91.6896,B 24.9464,C -1.6913,E1 24.9843,E2 354.628} C_DIS
LIN {X -9.2789,Y 126.6637,Z 140,A 89.7699,B 24.9464,C -1.6927,E1 24.9897,E2 356.5451} C_DIS
LIN {X -5.3953,Y 126.8893,Z 140,A 87.9977,B 24.9464,C -1.6925,E1 24.9946,E2 358.3183} C_DIS
LIN {X -2.1947,Y 126.9843,Z 140,A 86.609,B 24.9461,C -1.6956,E1 24.9985,E2 359.6999} C_DIS
LIN {X 1.5913,Y 126.9943,Z 140,A 84.7987,B 24.9464,C -1.6909,E1 25.0036,E2 361.521} C_DIS
LIN {X 5.6022,Y 126.8812,Z 140,A 82.9597,B 24.9464,C -1.6897,E1 25.0087,E2 363.3625} C_DIS
LIN {X 9.413,Y 126.6539,Z 140,A 81.3362,B 24.9462,C -1.6944,E1 25.0132,E2 364.974} C_DIS
LIN {X 13.3633,Y 126.2983,Z 140,A 79.5501,B 24.9462,C -1.6944,E1 25.0181,E2 366.7592} C_DIS
LIN {X 17.1849,Y 125.8369,Z 140,A 77.6897,B 24.9466,C -1.6879,E1 25.0233,E2 368.6334} C_DIS
LIN {X 20.9782,Y 125.2584,Z 140,A 76.0848,B 24.9463,C -1.6935,E1 25.0277,E2 370.2233} C_DIS
LIN {X 24.9619,Y 124.5263,Z 140,A 74.3701,B 24.946,C -1.6983,E1 25.0324,E2 371.9248} C_DIS
LIN {X 27.8437,Y 123.914,Z 140,A 72.9401,B 24.9463,C -1.6926,E1 25.0363,E2 373.3663} C_DIS
LIN {X 31.0546,Y 123.1478,Z 140,A 71.4458,B 24.9463,C -1.6915,E1 25.0404,E2 374.8611} C_DIS
LIN {X 34.586,Y 122.2035,Z 140,A 69.7275,B 24.9467,C -1.687,E1 25.045,E2 376.5873} C_DIS
LIN {X 38.1768,Y 121.1301,Z 140,A 68.2657,B 24.946,C -1.697,E1 25.0489,E2 378.0229} C_DIS
LIN {X 42.3724,Y 119.7282,Z 140,A 64.8905,B 24.9504,C -1.6277,E1 25.0582,E2 381.5551} C_DIS
LIN {X 49.676,Y 116.8871,Z 140,A 62.4594,B 24.9472,C -1.6779,E1 25.0641,E2 383.8619} C_DIS
LIN {X 53.1833,Y 115.331,Z 140,A 60.9347,B 24.9467,C -1.6862,E1 25.0679,E2 385.3633} C_DIS
LIN {X 55.9821,Y 113.9988,Z 140,A 59.2984,B 24.9476,C -1.6726,E1 25.0721,E2 387.0274} C_DIS
LIN {X 60.4466,Y 111.6983,Z 140,A 57.0917,B 24.9476,C -1.6724,E1 25.0775,E2 389.2283} C_DIS
LIN {X 64.0544,Y 109.669,Z 140,A 55.0728,B 24.9482,C -1.6621,E1 25.0825,E2 391.2655} C_DIS
LIN {X 68.5637,Y 106.9074,Z 140,A 52.8875,B 24.9478,C -1.6683,E1 25.0876,E2 393.429} C_DIS
LIN {X 72.2162,Y 104.4755,Z 140,A 50.9379,B 24.948,C -1.6665,E1 25.0921,E2 395.3763} C_DIS
LIN {X 75.7912,Y 101.911,Z 140,A 49.0314,B 24.948,C -1.667,E1 25.0964,E2 397.2751} C_DIS
LIN {X 82.3529,Y 96.6859,Z 140,A 45.1793,B 24.9486,C -1.6563,E1 25.1048,E2 401.1379} C_DIS
LIN {X 85.5316,Y 93.8859,Z 140,A 43.3035,B 24.9487,C -1.6541,E1 25.1087,E2 403.0113} C_DIS
LIN {X 88.6412,Y 90.9563,Z 140,A 41.3054,B 24.9492,C -1.6464,E1 25.1127,E2 405.0193} C_DIS
LIN {X 91.7154,Y 87.8548,Z 140,A 39.3795,B 24.9493,C -1.6443,E1 25.1165,E2 406.9418} C_DIS
LIN {X 94.826,Y 84.4884,Z 140,A 37.312,B 24.9496,C -1.6396,E1 25.1204,E2 409.0114} C_DIS
LIN {X 97.6518,Y 81.2056,Z 140,A 35.3626,B 24.9499,C -1.6352,E1 25.1239,E2 410.9623} C_DIS
LIN {X 99.9337,Y 78.3799,Z 140,A 33.7626,B 24.95,C -1.6331,E1 25.1266,E2 412.5596} C_DIS
LIN {X 101.7424,Y 76.0177,Z 140,A 31.7326,B 24.9523,C -1.5947,E1 25.1302,E2 414.6705} C_DIS
LIN {X 104.9869,Y 71.4704,Z 140,A 29.886,B 24.9507,C -1.6225,E1 25.133,E2 416.4425} C_DIS
LIN {X 107.3723,Y 67.8332,Z 140,A 27.9718,B 24.9508,C -1.6198,E1 25.1359,E2 418.3535} C_DIS
LIN {X 109.0837,Y 65.0454,Z 140,A 26.3384,B 24.9516,C -1.6076,E1 25.1382,E2 420.0072} C_DIS
LIN {X 111.6931,Y 60.4562,Z 140,A 24.0828,B 24.9516,C -1.6076,E1 25.1413,E2 422.2514} C_DIS
LIN {X 113.2997,Y 57.384,Z 140,A 22.3495,B 24.9524,C -1.5944,E1 25.1435,E2 424.0063} C_DIS
LIN {X 114.7456,Y 54.4356,Z 140,A 21.0992,B 24.9519,C -1.602,E1 25.145,E2 425.232} C_DIS
LIN {X 116.5422,Y 50.4737,Z 140,A 19.2589,B 24.9519,C -1.6026,E1 25.1471,E2 427.0607} C_DIS
LIN {X 117.7813,Y 47.5107,Z 140,A 17.8381,B 24.952,C -1.5998,E1 25.1486,E2 428.4805} C_DIS
LIN {X 119.3118,Y 43.5272,Z 140,A 16.037,B 24.952,C -1.6005,E1 25.1503,E2 430.27} C_DIS
LIN {X 121.7783,Y 36.0544,Z 140,A 12.2025,B 24.9535,C -1.5747,E1 25.1537,E2 434.1434} C_DIS
LIN {X 122.9133,Y 31.9784,Z 140,A 10.3537,B 24.9537,C -1.5718,E1 25.155,E2 435.9883} C_DIS
LIN {X 123.7835,Y 28.4148,Z 140,A 8.6931,B 24.954,C -1.5664,E1 25.1561,E2 437.6522} C_DIS
LIN {X 124.7163,Y 23.9921,Z 140,A 6.7831,B 24.954,C -1.5666,E1 25.1571,E2 439.5506} C_DIS
LIN {X 125.3593,Y 20.3737,Z 140,A 5.0322,B 24.9546,C -1.5564,E1 25.1579,E2 441.3152} C_DIS
LIN {X 125.9401,Y 16.3971,Z 140,A 3.3443,B 24.9546,C -1.5571,E1 25.1586,E2 442.9915} C_DIS
LIN {X 126.3794,Y 12.5793,Z 140,A 1.5645,B 24.955,C -1.549,E1 25.1591,E2 444.7798} C_DIS
LIN {X 126.6938,Y 8.8665,Z 140,A -0.1426,B 24.9554,C -1.5422,E1 25.1595,E2 446.4929} C_DIS
LIN {X 126.91,Y 4.8653,Z 140,A -1.856,B 24.9554,C -1.5412,E1 25.1597,E2 448.1985} C_DIS
LIN {X 127.0041,Y 0.5399,Z 140,A -3.791,B 24.9558,C -1.5356,E1 25.1597,E2 450.135} C_DIS
LIN {X 126.9596,Y -3.3314,Z 140,A -5.5285,B 24.9561,C -1.5304,E1 25.1597,E2 451.8746} C_DIS
LIN {X 126.8084,Y -7.0653,Z 140,A -7.2859,B 24.9567,C -1.521,E1 25.1595,E2 453.6435} C_DIS
LIN {X 126.5443,Y -10.7862,Z 140,A -8.8794,B 24.9567,C -1.5202,E1 25.1591,E2 455.2296} C_DIS
LIN {X 126.1426,Y -14.7614,Z 140,A -10.6683,B 24.957,C -1.515,E1 25.1586,E2 457.0203} C_DIS
LIN {X 125.6913,Y -18.2077,Z 140,A -12.2558,B 24.9574,C -1.5088,E1 25.158,E2 458.6129} C_DIS
LIN {X 125.0679,Y -22.0878,Z 140,A -14.0052,B 24.9576,C -1.5042,E1 25.1572,E2 460.3628} C_DIS
LIN {X 124.3845,Y -25.6588,Z 140,A -15.8991,B 24.9587,C -1.4856,E1 25.1561,E2 462.2896} C_DIS
LIN {X 123.6778,Y -28.8777,Z 140,A -17.1846,B 24.9583,C -1.4912,E1 25.1553,E2 463.5544} C_DIS
LIN {X 122.7456,Y -32.6077,Z 140,A -18.8114,B 24.9583,C -1.4912,E1 25.1542,E2 465.1717} C_DIS
LIN {X 121.647,Y -36.4991,Z 140,A -20.8591,B 24.9593,C -1.4737,E1 25.1526,E2 467.2492} C_DIS
LIN {X 120.1548,Y -41.1431,Z 140,A -22.8297,B 24.959,C -1.4787,E1 25.1508,E2 469.1968} C_DIS
LIN {X 118.5973,Y -45.4396,Z 140,A -24.9204,B 24.9595,C -1.4706,E1 25.1488,E2 471.2948} C_DIS
LIN {X 117.1901,Y -48.9506,Z 140,A -26.5715,B 24.9596,C -1.4682,E1 25.1471,E2 472.9425} C_DIS
LIN {X 115.7047,Y -52.367,Z 140,A -28.6311,B 24.961,C -1.4432,E1 25.1447,E2 475.0498} C_DIS
LIN {X 114.0784,Y -55.8208,Z 140,A -29.9193,B 24.96,C -1.4605,E1 25.1431,E2 476.2902} C_DIS
LIN {X 112.4775,Y -58.9786,Z 140,A -31.4529,B 24.9601,C -1.459,E1 25.1412,E2 477.8192} C_DIS
LIN {X 110.5244,Y -62.5673,Z 140,A -33.4622,B 24.9609,C -1.4448,E1 25.1384,E2 479.8516} C_DIS
LIN {X 108.2317,Y -66.4534,Z 140,A -35.4358,B 24.961,C -1.4421,E1 25.1356,E2 481.8215} C_DIS
LIN {X 105.9395,Y -70.0502,Z 140,A -37.0629,B 24.9605,C -1.452,E1 25.1332,E2 483.4171} C_DIS
LIN {X 102.3234,Y -75.2334,Z 140,A -39.9356,B 24.961,C -1.4428,E1 25.1286,E2 486.2976} C_DIS
LIN {X 99.7673,Y -78.5917,Z 140,A -41.9672,B 24.9616,C -1.4309,E1 25.1251,E2 488.3476} C_DIS
LIN {X 97.2506,Y -81.6852,Z 140,A -44.151,B 24.963,C -1.4061,E1 25.1211,E2 490.5797} C_DIS
LIN {X 94.93,Y -84.3715,Z 140,A -45.4841,B 24.9625,C -1.4158,E1 25.1187,E2 491.8841} C_DIS
LIN {X 92.0519,Y -87.5026,Z 140,A -47.411,B 24.9627,C -1.4104,E1 25.115,E2 493.8151} C_DIS
LIN {X 89.8134,Y -89.799,Z 140,A -48.8798,B 24.963,C -1.4057,E1 25.1121,E2 495.2889} C_DIS
LIN {X 85.9065,Y -93.5426,Z 140,A -51.2375,B 24.963,C -1.4041,E1 25.1073,E2 497.6407} C_DIS
LIN {X 82.5695,Y -96.5018,Z 140,A -53.2767,B 24.9634,C -1.398,E1 25.103,E2 499.6863} C_DIS
LIN {X 80.0303,Y -98.6177,Z 140,A -54.6501,B 24.9633,C -1.4006,E1 25.1001,E2 501.0482} C_DIS
LIN {X 75.5158,Y -102.116,Z 140,A -57.319,B 24.9638,C -1.3903,E1 25.0941,E2 503.7318} C_DIS
LIN {X 70.814,Y -105.4306,Z 140,A -60.2452,B 24.9649,C -1.368,E1 25.0873,E2 506.7006} C_DIS
LIN {X 67.4743,Y -107.5989,Z 140,A -61.6799,B 24.9642,C -1.3829,E1 25.084,E2 508.0955} C_DIS
LIN {X 63.8308,Y -109.7991,Z 140,A -63.5744,B 24.9642,C -1.3806,E1 25.0795,E2 509.9895} C_DIS
LIN {X 60.0695,Y -111.9009,Z 140,A -65.5939,B 24.9647,C -1.3733,E1 25.0745,E2 512.0204} C_DIS
LIN {X 56.3585,Y -113.8131,Z 140,A -67.2954,B 24.9644,C -1.3794,E1 25.0703,E2 513.7029} C_DIS
LIN {X 53.6678,Y -115.107,Z 140,A -68.664,B 24.9645,C -1.3761,E1 25.0668,E2 515.0757} C_DIS
LIN {X 50.4459,Y -116.5543,Z 140,A -70.0583,B 24.9641,C -1.3838,E1 25.0633,E2 516.4485} C_DIS
LIN {X 45.4928,Y -118.5766,Z 140,A -72.386,B 24.9641,C -1.3846,E1 25.0573,E2 518.7689} C_DIS
LIN {X 38.3109,Y -121.0872,Z 140,A -76.0765,B 24.965,C -1.367,E1 25.0475,E2 522.4937} C_DIS
LIN {X 33.2562,Y -122.5726,Z 140,A -78.515,B 24.9653,C -1.3612,E1 25.0409,E2 524.9418} C_DIS
LIN {X 29.7908,Y -123.4595,Z 140,A -80.0324,B 24.9651,C -1.3644,E1 25.0368,E2 526.4494} C_DIS
LIN {X 26.3037,Y -124.2502,Z 140,A -81.6268,B 24.9651,C -1.3638,E1 25.0325,E2 528.0431} C_DIS
LIN {X 22.5358,Y -124.9877,Z 140,A -83.3772,B 24.9653,C -1.3615,E1 25.0277,E2 529.7971} C_DIS
LIN {X 19.5295,Y -125.4925,Z 140,A -84.7503,B 24.9653,C -1.3605,E1 25.0239,E2 531.171} C_DIS
LIN {X 15.9183,Y -126.0029,Z 140,A -86.5185,B 24.9657,C -1.3533,E1 25.0189,E2 532.9549} C_DIS
LIN {X 12.0316,Y -126.4319,Z 140,A -88.1987,B 24.9655,C -1.3565,E1 25.0143,E2 534.6264} C_DIS
LIN {X 7.9194,Y -126.756,Z 140,A -90.0221,B 24.9655,C -1.3575,E1 25.0092,E2 536.4466} C_DIS
LIN {X 4.119,Y -126.9378,Z 140,A -91.8474,B 24.9658,C -1.3515,E1 25.0041,E2 538.2857} C_DIS
LIN {X 0.8984,Y -126.9978,Z 140,A -92.7208,B 24.9643,C -1.3799,E1 25.0019,E2 539.0917} C_DIS
Enddeposition()
LIN {X 0.8984,Y -126.9978,Z 140,A -92.7208,B 24.9643,C -1.3799,E1 25.0019,E2 539.0917} C_DIS
Startdeposition()
$VEL.CP = VEL_PRINT
LIN {X 2.3032,Y -126.0074,Z 140,A -91.7748,B 24.8764,C -1.3939,E1 24.9175,E2 538.1004} C_DIS
LIN {X 6.3467,Y -125.8683,Z 140,A -90.0181,B 24.8766,C -1.3905,E1 24.9224,E2 536.3524} C_DIS
LIN {X 10.3379,Y -125.6037,Z 140,A -88.1492,B 24.8764,C -1.3938,E1 24.9276,E2 534.4764} C_DIS
LIN {X 14.5036,Y -125.1915,Z 140,A -86.2599,B 24.8764,C -1.3943,E1 24.9329,E2 532.5874} C_DIS
LIN {X 18.1497,Y -124.7147,Z 140,A -84.5151,B 24.8761,C -1.3991,E1 24.9377,E2 530.8327} C_DIS
LIN {X 22.3739,Y -124.0262,Z 140,A -82.6856,B 24.8763,C -1.3948,E1 24.9427,E2 529.0154} C_DIS
LIN {X 27.0103,Y -123.1002,Z 140,A -80.4311,B 24.876,C -1.402,E1 24.9489,E2 526.7466} C_DIS
LIN {X 31.0127,Y -122.1526,Z 140,A -78.6415,B 24.876,C -1.3998,E1 24.9538,E2 524.9647} C_DIS
LIN {X 37.361,Y -120.3637,Z 140,A -75.8069,B 24.8763,C -1.3949,E1 24.9614,E2 522.1466} C_DIS
LIN {X 41.5032,Y -118.9981,Z 140,A -73.3688,B 24.875,C -1.4205,E1 24.9679,E2 519.6525} C_DIS
LIN {X 44.814,Y -117.7927,Z 140,A -72.1948,B 24.876,C -1.4009,E1 24.9709,E2 518.5275} C_DIS
LIN {X 48.9105,Y -116.1503,Z 140,A -70.1829,B 24.8759,C -1.4042,E1 24.9761,E2 516.5126} C_DIS
LIN {X 51.5813,Y -114.9886,Z 140,A -68.8017,B 24.8756,C -1.4091,E1 24.9796,E2 515.123} C_DIS
LIN {X 54.4656,Y -113.6508,Z 140,A -67.3625,B 24.8755,C -1.4111,E1 24.9833,E2 513.6827} C_DIS
LIN {X 57.3457,Y -112.2251,Z 140,A -65.909,B 24.8754,C -1.4132,E1 24.9869,E2 512.2284} C_DIS
LIN {X 60.6405,Y -110.4821,Z 140,A -64.0963,B 24.8749,C -1.4222,E1 24.9914,E2 510.3995} C_DIS
LIN {X 64.25,Y -108.4228,Z 140,A -62.3082,B 24.8749,C -1.4205,E1 24.9957,E2 508.6209} C_DIS
LIN {X 67.7038,Y -106.3002,Z 140,A -60.4567,B 24.8748,C -1.4245,E1 25.0001,E2 506.7658} C_DIS
LIN {X 71.5834,Y -103.7262,Z 140,A -58.0768,B 24.8738,C -1.4424,E1 25.0057,E2 504.3515} C_DIS
LIN {X 74.3054,Y -101.7954,Z 140,A -57.0687,B 24.875,C -1.4194,E1 25.0078,E2 503.4016} C_DIS
LIN {X 79.8756,Y -97.4852,Z 140,A -53.8953,B 24.8747,C -1.4249,E1 25.0148,E2 500.2268} C_DIS
LIN {X 83.1518,Y -94.7068,Z 140,A -51.6448,B 24.8737,C -1.4447,E1 25.0197,E2 497.9382} C_DIS
LIN {X 88.6176,Y -89.6128,Z 140,A -48.4499,B 24.8737,C -1.4425,E1 25.0261,E2 494.7618} C_DIS
LIN {X 92.5162,Y -85.5825,Z 140,A -45.8695,B 24.8734,C -1.4505,E1 25.0311,E2 492.1736} C_DIS
LIN {X 95.964,Y -81.6965,Z 140,A -43.3322,B 24.8725,C -1.4659,E1 25.0358,E2 489.6115} C_DIS
LIN {X 98.8232,Y -78.2144,Z 140,A -41.4999,B 24.8728,C -1.4601,E1 25.039,E2 487.8013} C_DIS
LIN {X 101.1351,Y -75.2007,Z 140,A -39.6831,B 24.8723,C -1.4696,E1 25.042,E2 485.9709} C_DIS
LIN {X 103.925,Y -71.2955,Z 140,A -37.5141,B 24.872,C -1.4751,E1 25.0455,E2 483.7995} C_DIS
LIN {X 105.5752,Y -68.8287,Z 140,A -36.1144,B 24.8716,C -1.4816,E1 25.0477,E2 482.3914} C_DIS
LIN {X 107.9274,Y -65.0781,Z 140,A -34.1675,B 24.8716,C -1.484,E1 25.0505,E2 480.4487} C_DIS
LIN {X 110.0192,Y -61.4762,Z 140,A -32.2357,B 24.8711,C -1.4916,E1 25.0532,E2 478.509} C_DIS
LIN {X 112.1467,Y -57.4998,Z 140,A -30.2759,B 24.8711,C -1.4931,E1 25.0557,E2 476.556} C_DIS
LIN {X 114.3362,Y -53.0116,Z 140,A -27.8752,B 24.8702,C -1.5069,E1 25.0587,E2 474.1357} C_DIS
LIN {X 116.0563,Y -49.1357,Z 140,A -26.2257,B 24.8707,C -1.4983,E1 25.0605,E2 472.5157} C_DIS
LIN {X 117.5797,Y -45.3663,Z 140,A -24.2983,B 24.8701,C -1.5082,E1 25.0625,E2 470.5754} C_DIS
LIN {X 119.8344,Y -39.0287,Z 140,A -20.698,B 24.8679,C -1.5465,E1 25.0658,E2 466.9051} C_DIS
LIN {X 121.1386,Y -34.7694,Z 140,A -19.3037,B 24.8695,C -1.5197,E1 25.0668,E2 465.5819} C_DIS
LIN {X 121.8376,Y -32.2289,Z 140,A -17.9774,B 24.8689,C -1.5304,E1 25.0678,E2 464.2382} C_DIS
LIN {X 123.5271,Y -24.9825,Z 140,A -14.685,B 24.8685,C -1.5366,E1 25.0698,E2 460.9503} C_DIS
LIN {X 124.2703,Y -20.9767,Z 140,A -12.8374,B 24.8682,C -1.5424,E1 25.0707,E2 459.0997} C_DIS
LIN {X 124.7977,Y -17.5689,Z 140,A -11.2121,B 24.8677,C -1.5506,E1 25.0714,E2 457.4648} C_DIS
LIN {X 125.3174,Y -13.3662,Z 140,A -9.4616,B 24.8679,C -1.5478,E1 25.0719,E2 455.7313} C_DIS
LIN {X 125.6142,Y -10.2133,Z 140,A -7.979,B 24.8675,C -1.5547,E1 25.0723,E2 454.241} C_DIS
LIN {X 125.8692,Y -6.3283,Z 140,A -6.1801,B 24.867,C -1.5621,E1 25.0726,E2 452.4355} C_DIS
LIN {X 126.0078,Y -2.2782,Z 140,A -4.3442,B 24.8667,C -1.5678,E1 25.0727,E2 450.5969} C_DIS
LIN {X 126.0129,Y 1.9732,Z 140,A -2.46,B 24.8665,C -1.5716,E1 25.0727,E2 448.715} C_DIS
LIN {X 125.9049,Y 5.6172,Z 140,A -0.6821,B 24.8658,C -1.5833,E1 25.0725,E2 446.9201} C_DIS
LIN {X 125.6711,Y 9.4858,Z 140,A 1.0626,B 24.8655,C -1.5882,E1 25.0721,E2 445.1742} C_DIS
LIN {X 125.2759,Y 13.7518,Z 140,A 2.9904,B 24.8652,C -1.5935,E1 25.0716,E2 443.2454} C_DIS
LIN {X 124.7606,Y 17.8289,Z 140,A 4.7401,B 24.8652,C -1.5933,E1 25.071,E2 441.5064} C_DIS
LIN {X 124.134,Y 21.7714,Z 140,A 6.5936,B 24.8647,C -1.6012,E1 25.0701,E2 439.6454} C_DIS
LIN {X 123.5111,Y 25.0614,Z 140,A 8.0365,B 24.8647,C -1.6019,E1 25.0693,E2 438.2093} C_DIS
LIN {X 122.6513,Y 28.9829,Z 140,A 9.7481,B 24.8647,C -1.6017,E1 25.0683,E2 436.5081} C_DIS
LIN {X 121.5641,Y 33.2522,Z 140,A 12.3051,B 24.8625,C -1.6369,E1 25.0664,E2 433.8826} C_DIS
LIN {X 120.5041,Y 36.9024,Z 140,A 13.7286,B 24.8632,C -1.6263,E1 25.0653,E2 432.4922} C_DIS
LIN {X 118.6468,Y 42.4972,Z 140,A 15.9949,B 24.864,C -1.6129,E1 25.0633,E2 430.2704} C_DIS
LIN {X 117.6365,Y 45.2204,Z 140,A 17.6204,B 24.8628,C -1.6327,E1 25.0616,E2 428.6072} C_DIS
LIN {X 116.2988,Y 48.5549,Z 140,A 19.1374,B 24.8628,C -1.6315,E1 25.06,E2 427.1014} C_DIS
LIN {X 115.0332,Y 51.4815,Z 140,A 20.6228,B 24.8625,C -1.6376,E1 25.0584,E2 425.6098} C_DIS
LIN {X 113.6478,Y 54.4718,Z 140,A 23.0263,B 24.8592,C -1.6892,E1 25.0553,E2 423.0972} C_DIS
LIN {X 110.7515,Y 60.1467,Z 140,A 25.6836,B 24.8595,C -1.6847,E1 25.0518,E2 420.4646} C_DIS
LIN {X 108.1836,Y 64.6513,Z 140,A 27.1798,B 24.8619,C -1.6464,E1 25.0498,E2 419.0667} C_DIS
LIN {X 106.4155,Y 67.5225,Z 140,A 28.9484,B 24.8609,C -1.6626,E1 25.0472,E2 417.2687} C_DIS
LIN {X 104.046,Y 71.1192,Z 140,A 31.293,B 24.8593,C -1.6878,E1 25.0434,E2 414.8762} C_DIS
LIN {X 101.6409,Y 74.5158,Z 140,A 32.4703,B 24.8614,C -1.6557,E1 25.0416,E2 413.7805} C_DIS
LIN {X 99.8495,Y 76.9005,Z 140,A 34.1467,B 24.8601,C -1.6755,E1 25.0387,E2 412.0652} C_DIS
LIN {X 97.1306,Y 80.3063,Z 140,A 36.0876,B 24.8599,C -1.6782,E1 25.0353,E2 410.1269} C_DIS
LIN {X 94.2148,Y 83.7086,Z 140,A 38.1183,B 24.8597,C -1.6827,E1 25.0316,E2 408.0949} C_DIS
LIN {X 91.3409,Y 86.8355,Z 140,A 40.0693,B 24.8593,C -1.6881,E1 25.0279,E2 406.1396} C_DIS
LIN {X 88.1196,Y 90.1022,Z 140,A 42.0658,B 24.8593,C -1.6881,E1 25.0239,E2 404.1517} C_DIS
LIN {X 85.0018,Y 93.0499,Z 140,A 44.0813,B 24.8588,C -1.6954,E1 25.0198,E2 402.1269} C_DIS
LIN {X 81.7261,Y 95.9391,Z 140,A 46.1689,B 24.8583,C -1.7046,E1 25.0153,E2 400.0259} C_DIS
LIN {X 76.835,Y 99.8997,Z 140,A 48.6473,B 24.8592,C -1.6906,E1 25.01,E2 397.59} C_DIS
LIN {X 74.2712,Y 101.8202,Z 140,A 50.3756,B 24.8581,C -1.7069,E1 25.0061,E2 395.8292} C_DIS
LIN {X 70.4557,Y 104.4964,Z 140,A 52.4749,B 24.8579,C -1.7095,E1 25.0012,E2 393.7309} C_DIS
LIN {X 66.9452,Y 106.7799,Z 140,A 54.358,B 24.8579,C -1.7115,E1 24.9968,E2 391.8492} C_DIS
LIN {X 59.9233,Y 110.8727,Z 140,A 57.8257,B 24.8582,C -1.7055,E1 24.9885,E2 388.4062} C_DIS
LIN {X 55.1715,Y 113.3116,Z 140,A 60.3126,B 24.8578,C -1.7115,E1 24.9823,E2 385.9117} C_DIS
LIN {X 52.6376,Y 114.5091,Z 140,A 61.6483,B 24.8575,C -1.7161,E1 24.9788,E2 384.5686} C_DIS
LIN {X 48.6404,Y 116.2631,Z 140,A 63.9204,B 24.8564,C -1.7327,E1 24.9729,E2 382.2627} C_DIS
LIN {X 45.6241,Y 117.4795,Z 140,A 65.3858,B 24.8564,C -1.7335,E1 24.9691,E2 380.7985} C_DIS
LIN {X 42.6174,Y 118.6034,Z 140,A 66.4913,B 24.8574,C -1.7173,E1 24.9663,E2 379.7338} C_DIS
LIN {X 39.4162,Y 119.7061,Z 140,A 68.2113,B 24.8568,C -1.7276,E1 24.9617,E2 377.9927} C_DIS
LIN {X 35.4299,Y 120.9452,Z 140,A 69.9623,B 24.8572,C -1.7218,E1 24.9571,E2 376.2587} C_DIS
LIN {X 32.1743,Y 121.8521,Z 140,A 71.477,B 24.8572,C -1.7218,E1 24.953,E2 374.7465} C_DIS
LIN {X 28.8108,Y 122.6928,Z 140,A 73.3902,B 24.856,C -1.7392,E1 24.9477,E2 372.7945} C_DIS
LIN {X 22.9512,Y 123.9227,Z 140,A 75.9226,B 24.8565,C -1.731,E1 24.9408,E2 370.2844} C_DIS
LIN {X 19.1632,Y 124.5627,Z 140,A 77.54,B 24.8569,C -1.7253,E1 24.9364,E2 368.6823} C_DIS
LIN {X 15.1914,Y 125.1094,Z 140,A 79.3889,B 24.8569,C -1.727,E1 24.9313,E2 366.8308} C_DIS
LIN {X 11.3416,Y 125.5187,Z 140,A 81.2417,B 24.8565,C -1.7317,E1 24.9261,E2 364.9681} C_DIS
LIN {X 7.5531,Y 125.8018,Z 140,A 82.9197,B 24.8567,C -1.7294,E1 24.9214,E2 363.2963} C_DIS
LIN {X 3.4944,Y 125.9798,Z 140,A 84.7069,B 24.8569,C -1.7264,E1 24.9165,E2 361.5168} C_DIS
LIN {X -0.5087,Y 126.0274,Z 140,A 86.5489,B 24.8569,C -1.7271,E1 24.9113,E2 359.6731} C_DIS
LIN {X -3.7194,Y 125.9735,Z 140,A 88.0743,B 24.8566,C -1.7299,E1 24.907,E2 358.1411} C_DIS
LIN {X -7.8015,Y 125.7865,Z 140,A 89.86,B 24.8569,C -1.7257,E1 24.9021,E2 356.3647} C_DIS
LIN {X -11.8198,Y 125.4728,Z 140,A 91.7149,B 24.8569,C -1.7259,E1 24.8969,E2 354.5084} C_DIS
LIN {X -15.1808,Y 125.1107,Z 140,A 93.2954,B 24.8569,C -1.7271,E1 24.8925,E2 352.924} C_DIS
LIN {X -19.213,Y 124.5549,Z 140,A 95.06,B 24.8572,C -1.7218,E1 24.8877,E2 351.1706} C_DIS
LIN {X -22.8707,Y 123.9373,Z 140,A 96.8699,B 24.8569,C -1.7263,E1 24.8827,E2 349.348} C_DIS
LIN {X -28.6729,Y 122.7245,Z 140,A 99.9806,B 24.8557,C -1.7438,E1 24.8741,E2 346.1919} C_DIS
LIN {X -32.7485,Y 121.699,Z 140,A 101.3565,B 24.8575,C -1.7164,E1 24.8705,E2 344.8791} C_DIS
LIN {X -36.6799,Y 120.5722,Z 140,A 103.9393,B 24.8554,C -1.7486,E1 24.8634,E2 342.2151} C_DIS
LIN {X -41.5945,Y 118.9664,Z 140,A 105.6963,B 24.8574,C -1.7175,E1 24.859,E2 340.5289} C_DIS
LIN {X -45.3753,Y 117.5763,Z 140,A 107.4522,B 24.8578,C -1.7115,E1 24.8544,E2 338.7837} C_DIS
LIN {X -48.7929,Y 116.1994,Z 140,A 109.1364,B 24.8579,C -1.7096,E1 24.8501,E2 337.1003} C_DIS
LIN {X -54.5208,Y 113.6244,Z 140,A 111.9474,B 24.8584,C -1.7031,E1 24.843,E2 334.2979} C_DIS
LIN {X -57.7763,Y 112.006,Z 140,A 113.7576,B 24.8581,C -1.7076,E1 24.8384,E2 332.4719} C_DIS
LIN {X -64.4259,Y 108.3179,Z 140,A 116.9256,B 24.8593,C -1.688,E1 24.8308,E2 329.3414} C_DIS
LIN {X -67.0104,Y 106.7387,Z 140,A 118.6051,B 24.8586,C -1.6994,E1 24.8267,E2 327.6295} C_DIS
LIN {X -70.8872,Y 104.2044,Z 140,A 120.6827,B 24.8589,C -1.6939,E1 24.8219,E2 325.558} C_DIS
LIN {X -74.3577,Y 101.757,Z 140,A 122.5887,B 24.8593,C -1.6888,E1 24.8176,E2 323.6576} C_DIS
LIN {X -77.5597,Y 99.3382,Z 140,A 124.5055,B 24.8593,C -1.6891,E1 24.8133,E2 321.7331} C_DIS
LIN {X -80.9421,Y 96.6014,Z 140,A 126.4493,B 24.8596,C -1.6831,E1 24.8092,E2 319.7961} C_DIS
LIN {X -84.367,Y 93.6259,Z 140,A 128.5495,B 24.8598,C -1.68,E1 24.8048,E2 317.6949} C_DIS
LIN {X -87.4234,Y 90.7783,Z 140,A 130.4605,B 24.8601,C -1.676,E1 24.8009,E2 315.7856} C_DIS
LIN {X -90.5721,Y 87.6364,Z 140,A 132.4498,B 24.8605,C -1.6695,E1 24.797,E2 313.8033} C_DIS
LIN {X -93.4463,Y 84.5651,Z 140,A 134.3665,B 24.8608,C -1.6648,E1 24.7934,E2 311.8894} C_DIS
LIN {X -96.3008,Y 81.3005,Z 140,A 136.3976,B 24.8609,C -1.6624,E1 24.7897,E2 309.8548} C_DIS
LIN {X -99.0486,Y 77.9285,Z 140,A 138.3507,B 24.8613,C -1.656,E1 24.7863,E2 307.9078} C_DIS
LIN {X -101.7788,Y 74.328,Z 140,A 140.4019,B 24.8617,C -1.6502,E1 24.7829,E2 305.8605} C_DIS
LIN {X -104.028,Y 71.1455,Z 140,A 142.1948,B 24.862,C -1.6462,E1 24.78,E2 304.0684} C_DIS
LIN {X -106.3956,Y 67.554,Z 140,A 144.2059,B 24.8621,C -1.6431,E1 24.777,E2 302.0544} C_DIS
LIN {X -110.1253,Y 61.2857,Z 140,A 147.1897,B 24.8637,C -1.6183,E1 24.7728,E2 299.1145} C_DIS
LIN {X -112.097,Y 57.5974,Z 140,A 149.1959,B 24.8637,C -1.6173,E1 24.7702,E2 297.0999} C_DIS
LIN {X -113.0679,Y 55.6654,Z 140,A 151.1851,B 24.8611,C -1.6602,E1 24.7676,E2 294.9974} C_DIS
LIN {X -115.5551,Y 50.3002,Z 140,A 153.0434,B 24.8639,C -1.614,E1 24.7656,E2 293.2393} C_DIS
LIN {X -117.2551,Y 46.2015,Z 140,A 154.95,B 24.8646,C -1.6027,E1 24.7636,E2 291.349} C_DIS
LIN {X -118.6098,Y 42.5998,Z 140,A 156.8545,B 24.8646,C -1.6042,E1 24.7618,E2 289.4302} C_DIS
LIN {X -120.0884,Y 38.2334,Z 140,A 159.15,B 24.8644,C -1.6065,E1 24.7598,E2 287.1158} C_DIS
LIN {X -121.166,Y 34.6758,Z 140,A 160.8031,B 24.8648,C -1.5994,E1 24.7585,E2 285.4701} C_DIS
LIN {X -122.3099,Y 30.3926,Z 140,A 162.9464,B 24.8648,C -1.5987,E1 24.757,E2 283.316} C_DIS
LIN {X -123.5067,Y 25.0829,Z 140,A 165.1375,B 24.8661,C -1.5778,E1 24.7557,E2 281.1618} C_DIS
LIN {X -124.1966,Y 21.418,Z 140,A 166.9759,B 24.8661,C -1.5787,E1 24.7548,E2 279.3103} C_DIS
LIN {X -125.058,Y 15.6224,Z 140,A 169.5305,B 24.8669,C -1.565,E1 24.7538,E2 276.7731} C_DIS
LIN {X -125.5895,Y 10.5067,Z 140,A 171.6258,B 24.8679,C -1.5464,E1 24.7533,E2 274.7097} C_DIS
LIN {X -125.7888,Y 7.7639,Z 140,A 173.1902,B 24.8674,C -1.5565,E1 24.753,E2 273.1119} C_DIS
LIN {X -125.9742,Y 3.694,Z 140,A 175.6478,B 24.8661,C -1.5779,E1 24.7527,E2 270.5883} C_DIS
LIN {X -126.0248,Y -1.0993,Z 140,A 177.1422,B 24.8683,C -1.5396,E1 24.7527,E2 269.1764} C_DIS
LIN {X -125.9657,Y -3.9996,Z 140,A 178.6571,B 24.8681,C -1.5441,E1 24.7529,E2 267.6415} C_DIS
LIN {X -125.7799,Y -7.9086,Z 140,A -179.6518,B 24.8686,C -1.5344,E1 24.7531,E2 265.9635} C_DIS
LIN {X -125.3467,Y -13.0933,Z 140,A -177.231,B 24.8689,C -1.5292,E1 24.7537,E2 263.5405} C_DIS
LIN {X -124.9129,Y -16.7325,Z 140,A -175.5308,B 24.8692,C -1.5253,E1 24.7543,E2 261.8393} C_DIS
LIN {X -123.994,Y -22.554,Z 140,A -172.9756,B 24.87,C -1.5111,E1 24.7555,E2 259.3028} C_DIS
LIN {X -122.9208,Y -27.8134,Z 140,A -170.3978,B 24.87,C -1.5096,E1 24.757,E2 256.7134} C_DIS
LIN {X -122.2256,Y -30.7249,Z 140,A -168.8402,B 24.8698,C -1.5143,E1 24.758,E2 255.1354} C_DIS
LIN {X -120.6829,Y -36.3181,Z 140,A -166.5257,B 24.8711,C -1.4914,E1 24.7598,E2 252.8623} C_DIS
LIN {X -119.665,Y -39.5396,Z 140,A -164.8126,B 24.8709,C -1.4948,E1 24.7613,E2 251.1313} C_DIS
LIN {X -118.438,Y -43.0764,Z 140,A -163.0759,B 24.8711,C -1.4912,E1 24.7629,E2 249.3931} C_DIS
LIN {X -116.9231,Y -47.0319,Z 140,A -161.2191,B 24.8716,C -1.4823,E1 24.7648,E2 247.5471} C_DIS
LIN {X -115.6881,Y -49.9926,Z 140,A -159.6791,B 24.8716,C -1.4818,E1 24.7665,E2 245.9999} C_DIS
LIN {X -114.2483,Y -53.2017,Z 140,A -158.1339,B 24.872,C -1.4747,E1 24.7683,E2 244.4631} C_DIS
LIN {X -112.1638,Y -57.4661,Z 140,A -155.9568,B 24.8723,C -1.4694,E1 24.771,E2 242.2869} C_DIS
LIN {X -110.5071,Y -60.5947,Z 140,A -154.2901,B 24.8724,C -1.4676,E1 24.7732,E2 240.6158} C_DIS
LIN {X -108.4395,Y -64.222,Z 140,A -152.3144,B 24.8725,C -1.4659,E1 24.776,E2 238.6337} C_DIS
LIN {X -105.6252,Y -68.7517,Z 140,A -150.0119,B 24.8732,C -1.4539,E1 24.7794,E2 236.3482} C_DIS
LIN {X -102.8366,Y -72.8571,Z 140,A -147.642,B 24.8732,C -1.4533,E1 24.7832,E2 233.968} C_DIS
LIN {X -100.5261,Y -76.0129,Z 140,A -145.8885,B 24.8735,C -1.4477,E1 24.7861,E2 232.2193} C_DIS
LIN {X -97.7757,Y -79.5202,Z 140,A -143.7906,B 24.8735,C -1.4461,E1 24.7897,E2 230.1153} C_DIS
LIN {X -94.844,Y -82.9946,Z 140,A -141.4937,B 24.8733,C -1.452,E1 24.794,E2 227.7938} C_DIS
LIN {X -92.5752,Y -85.5183,Z 140,A -140.4383,B 24.8747,C -1.4258,E1 24.7959,E2 226.7965} C_DIS
LIN {X -90.3818,Y -87.833,Z 140,A -138.7616,B 24.8743,C -1.4332,E1 24.7992,E2 225.0948} C_DIS
LIN {X -87.3459,Y -90.8531,Z 140,A -136.7728,B 24.8744,C -1.431,E1 24.8031,E2 223.103} C_DIS
LIN {X -84.2499,Y -93.7308,Z 140,A -134.8298,B 24.8746,C -1.428,E1 24.8071,E2 221.1591} C_DIS
LIN {X -81.084,Y -96.4824,Z 140,A -132.943,B 24.8748,C -1.4234,E1 24.8111,E2 219.2761} C_DIS
LIN {X -78.1339,Y -98.8872,Z 140,A -131.1879,B 24.8749,C -1.4213,E1 24.815,E2 217.5194} C_DIS
LIN {X -74.9188,Y -101.3448,Z 140,A -129.3126,B 24.875,C -1.4196,E1 24.8192,E2 215.6413} C_DIS
LIN {X -71.0152,Y -104.1174,Z 140,A -127.4335,B 24.876,C -1.4019,E1 24.8234,E2 213.798} C_DIS
LIN {X -68.4529,Y -105.8192,Z 140,A -125.1441,B 24.8738,C -1.4421,E1 24.829,E2 211.4055} C_DIS
LIN {X -64.0553,Y -108.5372,Z 140,A -123.4138,B 24.8756,C -1.4089,E1 24.833,E2 209.7489} C_DIS
LIN {X -60.3422,Y -110.6448,Z 140,A -121.4004,B 24.8756,C -1.4096,E1 24.8379,E2 207.7279} C_DIS
LIN {X -56.9715,Y -112.4157,Z 140,A -119.7945,B 24.876,C -1.4014,E1 24.8418,E2 206.1371} C_DIS
LIN {X -54.1015,Y -113.8247,Z 140,A -118.4076,B 24.8763,C -1.3965,E1 24.8453,E2 204.7584} C_DIS
LIN {X -51.5276,Y -115.0126,Z 140,A -116.7705,B 24.8755,C -1.4117,E1 24.8496,E2 203.0811} C_DIS
LIN {X -45.5956,Y -117.4906,Z 140,A -114.1726,B 24.8764,C -1.3931,E1 24.8562,E2 200.5218} C_DIS
LIN {X -42.5132,Y -118.641,Z 140,A -112.5136,B 24.8761,C -1.3996,E1 24.8606,E2 198.8439} C_DIS
LIN {X -39.0982,Y -119.812,Z 140,A -111.0328,B 24.8766,C -1.3904,E1 24.8645,E2 197.3822} C_DIS
LIN {X -35.1339,Y -121.0319,Z 140,A -109.103,B 24.8766,C -1.3912,E1 24.8697,E2 195.4472} C_DIS
LIN {X -31.2512,Y -122.092,Z 140,A -106.9892,B 24.8759,C -1.4039,E1 24.8755,E2 193.3} C_DIS
LIN {X -26.608,Y -123.1871,Z 140,A -105.07,B 24.8766,C -1.3907,E1 24.8806,E2 191.4099} C_DIS
LIN {X -22.4945,Y -124.0046,Z 140,A -103.1478,B 24.8766,C -1.3907,E1 24.8859,E2 189.4855} C_DIS
LIN {X -18.9543,Y -124.595,Z 140,A -101.596,B 24.8768,C -1.3863,E1 24.8901,E2 187.9428} C_DIS
LIN {X -15.3621,Y -125.0891,Z 140,A -99.8334,B 24.8765,C -1.3916,E1 24.8951,E2 186.1663} C_DIS
LIN {X -11.4406,Y -125.5092,Z 140,A -98.067,B 24.8765,C -1.3901,E1 24.9,E2 184.4025} C_DIS
LIN {X -7.7697,Y -125.7884,Z 140,A -96.4506,B 24.8767,C -1.3873,E1 24.9044,E2 182.7922} C_DIS
LIN {X -3.8406,Y -125.9702,Z 140,A -94.5718,B 24.8765,C -1.3919,E1 24.9097,E2 180.9019} C_DIS
LIN {X 0.4859,Y -126.0275,Z 140,A -92.665,B 24.8766,C -1.3894,E1 24.915,E2 179.0012} C_DIS
LIN {X 0.4859,Y -126.0275,Z 140,A -92.665,B 24.8766,C -1.3894,E1 24.915,E2 179.0012} C_DIS
Enddeposition()
LIN {X 0.8761,Y -125.0483,Z 140,A -92.4542,B 24.3074,C -1.2895,E1 24.3417,E2 178.9509} C_DIS
Startdeposition()
$VEL.CP = VEL_PRINT
LIN {X -3.2797,Y -125.0104,Z 140,A -94.9742,B 24.3089,C -1.2599,E1 24.3345,E2 181.5429} C_DIS
LIN {X -7.0578,Y -124.8555,Z 140,A -96.8046,B 24.3091,C -1.2552,E1 24.3293,E2 183.3853} C_DIS
LIN {X -11.228,Y -124.55,Z 140,A -98.7436,B 24.3091,C -1.2542,E1 24.3239,E2 185.3277} C_DIS
LIN {X -15.2644,Y -124.1189,Z 140,A -100.5701,B 24.3091,C -1.256,E1 24.3189,E2 187.1509} C_DIS
LIN {X -18.9661,Y -123.6066,Z 140,A -102.1732,B 24.3088,C -1.2615,E1 24.3145,E2 188.7419} C_DIS
LIN {X -22.4064,Y -123.0299,Z 140,A -103.8215,B 24.3088,C -1.2597,E1 24.3099,E2 190.3963} C_DIS
LIN {X -26.4302,Y -122.2281,Z 140,A -105.5858,B 24.3086,C -1.2659,E1 24.3051,E2 192.1476} C_DIS
LIN {X -29.2426,Y -121.5859,Z 140,A -107.2038,B 24.3092,C -1.2529,E1 24.3007,E2 193.7995} C_DIS
LIN {X -33.5974,Y -120.4552,Z 140,A -109.0588,B 24.3087,C -1.2637,E1 24.2957,E2 195.6311} C_DIS
LIN {X -36.381,Y -119.644,Z 140,A -110.4295,B 24.3087,C -1.2627,E1 24.292,E2 197.0066} C_DIS
LIN {X -40.3709,Y -118.3588,Z 140,A -112.2365,B 24.3084,C -1.2695,E1 24.2873,E2 198.8006} C_DIS
LIN {X -43.4079,Y -117.2783,Z 140,A -113.7172,B 24.3084,C -1.2707,E1 24.2834,E2 200.2815} C_DIS
LIN {X -46.0297,Y -116.2757,Z 140,A -115.6394,B 24.3097,C -1.2429,E1 24.2782,E2 202.2756} C_DIS
LIN {X -50.0959,Y -114.5812,Z 140,A -117.1342,B 24.3084,C -1.2689,E1 24.2745,E2 203.7108} C_DIS
Enddeposition()
END
